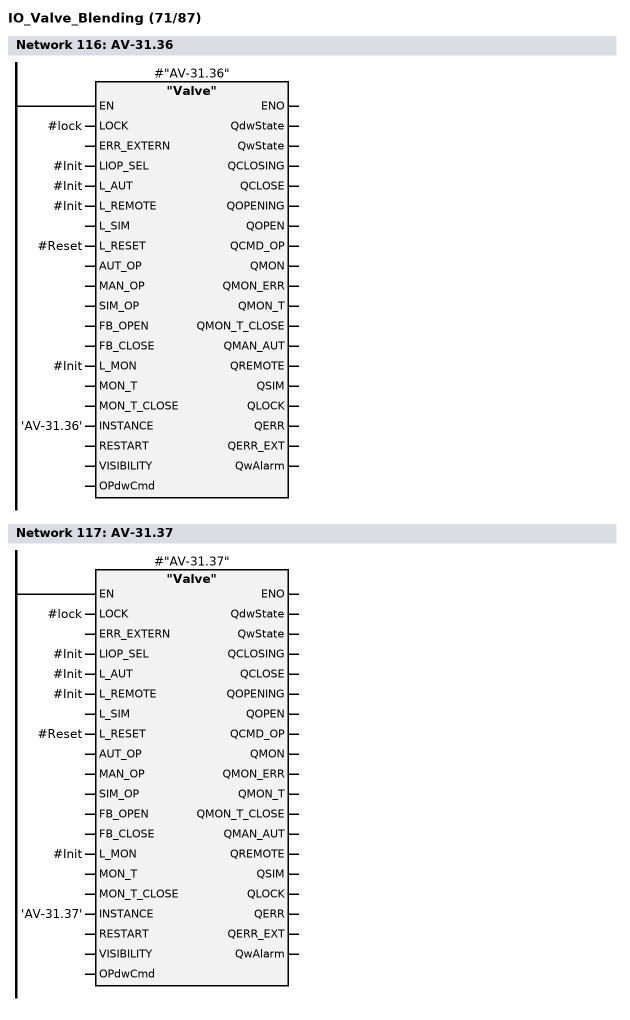
   RUNG wire#powerrail
      #"AV-31.36"(LOCK := #lock, ERR_EXTERN :=, LIOP_SEL := #Init, L_AUT := #Init, L_REMOTE := #Init, L_SIM :=, L_RESET := #Reset, AUT_OP :=, MAN_OP :=, SIM_OP :=, FB_OPEN :=, FB_CLOSE :=, L_MON := #Init, MON_T :=, MON_T_CLOSE :=, INSTANCE := 'AV-31.36', RESTART :=, VISIBILITY :=, OPdwCmd :=, QdwState =>, QwState =>, QCLOSING =>, QCLOSE =>, QOPENING =>, QOPEN =>, QCMD_OP =>, QMON =>, QMON_ERR =>, QMON_T =>, QMON_T_CLOSE =>, QMAN_AUT =>, QREMOTE =>, QSIM =>, QLOCK =>, QERR =>, QERR_EXT =>, QwAlarm =>)
   END_RUNG
   // the same network as SCL:
   #"AV-31.36"(LOCK := #lock,   // "Valve"
               LIOP_SEL := #Init,
               L_AUT := #Init,
               L_REMOTE := #Init,
               L_RESET := #Reset,
               L_MON := #Init,
               INSTANCE := 'AV-31.36');
END_REGION

REGION Network 117: AV-31.37
   RUNG wire#powerrail
      #"AV-31.37"(LOCK := #lock, ERR_EXTERN :=, LIOP_SEL := #Init, L_AUT := #Init, L_REMOTE := #Init, L_SIM :=, L_RESET := #Reset, AUT_OP :=, MAN_OP :=, SIM_OP :=, FB_OPEN :=, FB_CLOSE :=, L_MON := #Init, MON_T :=, MON_T_CLOSE :=, INSTANCE := 'AV-31.37', RESTART :=, VISIBILITY :=, OPdwCmd :=, QdwState =>, QwState =>, QCLOSING =>, QCLOSE =>, QOPENING =>, QOPEN =>, QCMD_OP =>, QMON =>, QMON_ERR =>, QMON_T =>, QMON_T_CLOSE =>, QMAN_AUT =>, QREMOTE =>, QSIM =>, QLOCK =>, QERR =>, QERR_EXT =>, QwAlarm =>)
   END_RUNG
   // the same network as SCL:
   #"AV-31.37"(LOCK := #lock,   // "Valve"
               LIOP_SEL := #Init,
               L_AUT := #Init,
               L_REMOTE := #Init,
               L_RESET := #Reset,
               L_MON := #Init,
               INSTANCE := 'AV-31.37');
END_REGION

REGION Network 118: AV-31.38
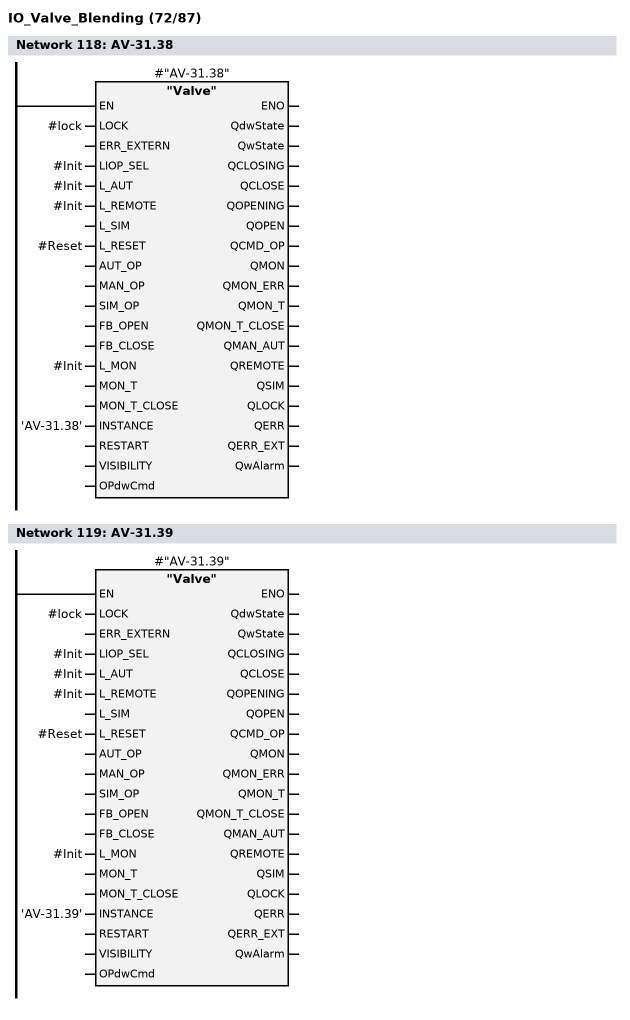
   RUNG wire#powerrail
      #"AV-31.38"(LOCK := #lock, ERR_EXTERN :=, LIOP_SEL := #Init, L_AUT := #Init, L_REMOTE := #Init, L_SIM :=, L_RESET := #Reset, AUT_OP :=, MAN_OP :=, SIM_OP :=, FB_OPEN :=, FB_CLOSE :=, L_MON := #Init, MON_T :=, MON_T_CLOSE :=, INSTANCE := 'AV-31.38', RESTART :=, VISIBILITY :=, OPdwCmd :=, QdwState =>, QwState =>, QCLOSING =>, QCLOSE =>, QOPENING =>, QOPEN =>, QCMD_OP =>, QMON =>, QMON_ERR =>, QMON_T =>, QMON_T_CLOSE =>, QMAN_AUT =>, QREMOTE =>, QSIM =>, QLOCK =>, QERR =>, QERR_EXT =>, QwAlarm =>)
   END_RUNG
   // the same network as SCL:
   #"AV-31.38"(LOCK := #lock,   // "Valve"
               LIOP_SEL := #Init,
               L_AUT := #Init,
               L_REMOTE := #Init,
               L_RESET := #Reset,
               L_MON := #Init,
               INSTANCE := 'AV-31.38');
END_REGION

REGION Network 119: AV-31.39
   RUNG wire#powerrail
      #"AV-31.39"(LOCK := #lock, ERR_EXTERN :=, LIOP_SEL := #Init, L_AUT := #Init, L_REMOTE := #Init, L_SIM :=, L_RESET := #Reset, AUT_OP :=, MAN_OP :=, SIM_OP :=, FB_OPEN :=, FB_CLOSE :=, L_MON := #Init, MON_T :=, MON_T_CLOSE :=, INSTANCE := 'AV-31.39', RESTART :=, VISIBILITY :=, OPdwCmd :=, QdwState =>, QwState =>, QCLOSING =>, QCLOSE =>, QOPENING =>, QOPEN =>, QCMD_OP =>, QMON =>, QMON_ERR =>, QMON_T =>, QMON_T_CLOSE =>, QMAN_AUT =>, QREMOTE =>, QSIM =>, QLOCK =>, QERR =>, QERR_EXT =>, QwAlarm =>)
   END_RUNG
   // the same network as SCL:
   #"AV-31.39"(LOCK := #lock,   // "Valve"
               LIOP_SEL := #Init,
               L_AUT := #Init,
               L_REMOTE := #Init,
               L_RESET := #Reset,
               L_MON := #Init,
               INSTANCE := 'AV-31.39');
END_REGION

REGION Network 120: AV-31.40
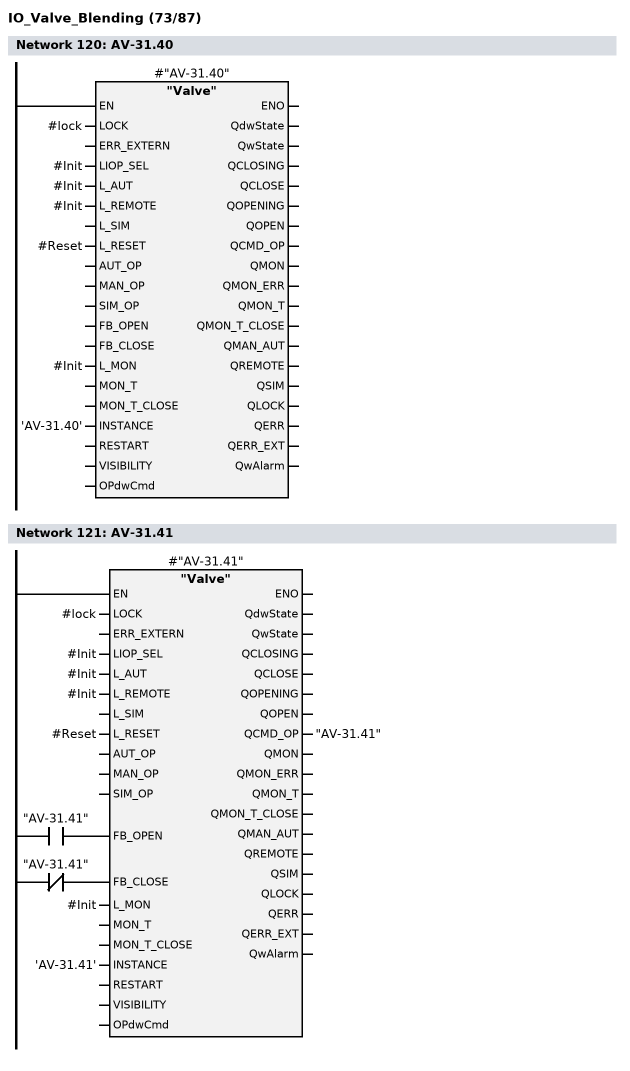
   RUNG wire#powerrail
      #"AV-31.40"(LOCK := #lock, ERR_EXTERN :=, LIOP_SEL := #Init, L_AUT := #Init, L_REMOTE := #Init, L_SIM :=, L_RESET := #Reset, AUT_OP :=, MAN_OP :=, SIM_OP :=, FB_OPEN :=, FB_CLOSE :=, L_MON := #Init, MON_T :=, MON_T_CLOSE :=, INSTANCE := 'AV-31.40', RESTART :=, VISIBILITY :=, OPdwCmd :=, QdwState =>, QwState =>, QCLOSING =>, QCLOSE =>, QOPENING =>, QOPEN =>, QCMD_OP =>, QMON =>, QMON_ERR =>, QMON_T =>, QMON_T_CLOSE =>, QMAN_AUT =>, QREMOTE =>, QSIM =>, QLOCK =>, QERR =>, QERR_EXT =>, QwAlarm =>)
   END_RUNG
   // the same network as SCL:
   #"AV-31.40"(LOCK := #lock,   // "Valve"
               LIOP_SEL := #Init,
               L_AUT := #Init,
               L_REMOTE := #Init,
               L_RESET := #Reset,
               L_MON := #Init,
               INSTANCE := 'AV-31.40');
END_REGION

REGION Network 121: AV-31.41
   RUNG wire#powerrail
      #"AV-31.41"(FB_OPEN := wire#w1, FB_CLOSE := wire#w2, LOCK := #lock, ERR_EXTERN :=, LIOP_SEL := #Init, L_AUT := #Init, L_REMOTE := #Init, L_SIM :=, L_RESET := #Reset, AUT_OP :=, MAN_OP :=, SIM_OP :=, L_MON := #Init, MON_T :=, MON_T_CLOSE :=, INSTANCE := 'AV-31.41', RESTART :=, VISIBILITY :=, OPdwCmd :=, QdwState =>, QwState =>, QCLOSING =>, QCLOSE =>, QOPENING =>, QOPEN =>, QCMD_OP => "AV-31.41", QMON =>, QMON_ERR =>, QMON_T =>, QMON_T_CLOSE =>, QMAN_AUT =>, QREMOTE =>, QSIM =>, QLOCK =>, QERR =>, QERR_EXT =>, QwAlarm =>)
   END_RUNG
   RUNG wire#powerrail
      Contact( "AV-31.41" )
   END_RUNG wire#w1
   RUNG wire#powerrail
      I_Contact( "AV-31.41" )
   END_RUNG wire#w2
   // the same network as SCL:
   #"AV-31.41"(LOCK := #lock,   // "Valve"
               LIOP_SEL := #Init,
               L_AUT := #Init,
               L_REMOTE := #Init,
               L_RESET := #Reset,
               FB_OPEN := "AV-31.41",
               FB_CLOSE := NOT "AV-31.41",
               L_MON := #Init,
               INSTANCE := 'AV-31.41',
               QCMD_OP => "AV-31.41");
END_REGION

REGION Network 122: AV-31.51
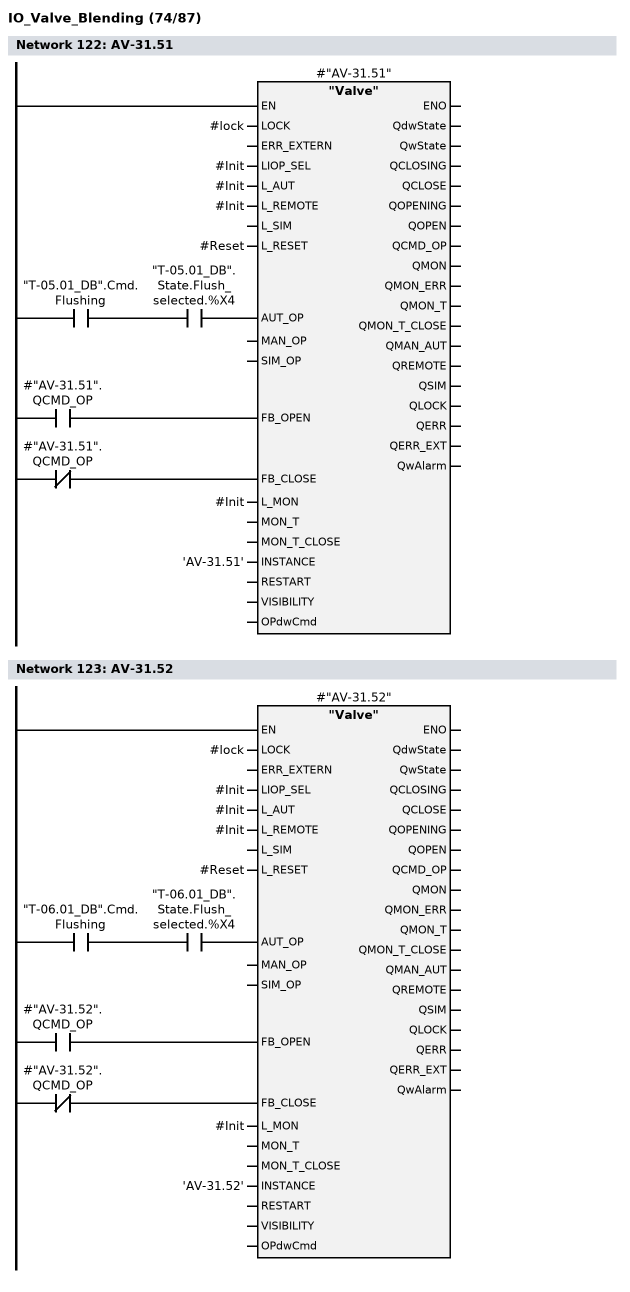
   RUNG wire#powerrail
      #"AV-31.51"(AUT_OP := wire#w1, FB_OPEN := wire#w2, FB_CLOSE := wire#w3, LOCK := #lock, ERR_EXTERN :=, LIOP_SEL := #Init, L_AUT := #Init, L_REMOTE := #Init, L_SIM :=, L_RESET := #Reset, MAN_OP :=, SIM_OP :=, L_MON := #Init, MON_T :=, MON_T_CLOSE :=, INSTANCE := 'AV-31.51', RESTART :=, VISIBILITY :=, OPdwCmd :=, QdwState =>, QwState =>, QCLOSING =>, QCLOSE =>, QOPENING =>, QOPEN =>, QCMD_OP =>, QMON =>, QMON_ERR =>, QMON_T =>, QMON_T_CLOSE =>, QMAN_AUT =>, QREMOTE =>, QSIM =>, QLOCK =>, QERR =>, QERR_EXT =>, QwAlarm =>)
   END_RUNG
   RUNG wire#powerrail
      Contact( "T-05.01_DB".Cmd.Flushing )
      Contact( "T-05.01_DB".State.Flush_selected.%X4 )
   END_RUNG wire#w1
   RUNG wire#powerrail
      Contact( #"AV-31.51".QCMD_OP )
   END_RUNG wire#w2
   RUNG wire#powerrail
      I_Contact( #"AV-31.51".QCMD_OP )
   END_RUNG wire#w3
   // the same network as SCL:
   #"AV-31.51"(LOCK := #lock,   // "Valve"
               LIOP_SEL := #Init,
               L_AUT := #Init,
               L_REMOTE := #Init,
               L_RESET := #Reset,
               AUT_OP := "T-05.01_DB".Cmd.Flushing AND "T-05.01_DB".State.Flush_selected.%X4,
               FB_OPEN := #"AV-31.51".QCMD_OP,
               FB_CLOSE := NOT #"AV-31.51".QCMD_OP,
               L_MON := #Init,
               INSTANCE := 'AV-31.51');
END_REGION

REGION Network 123: AV-31.52
   RUNG wire#powerrail
      #"AV-31.52"(AUT_OP := wire#w1, FB_OPEN := wire#w2, FB_CLOSE := wire#w3, LOCK := #lock, ERR_EXTERN :=, LIOP_SEL := #Init, L_AUT := #Init, L_REMOTE := #Init, L_SIM :=, L_RESET := #Reset, MAN_OP :=, SIM_OP :=, L_MON := #Init, MON_T :=, MON_T_CLOSE :=, INSTANCE := 'AV-31.52', RESTART :=, VISIBILITY :=, OPdwCmd :=, QdwState =>, QwState =>, QCLOSING =>, QCLOSE =>, QOPENING =>, QOPEN =>, QCMD_OP =>, QMON =>, QMON_ERR =>, QMON_T =>, QMON_T_CLOSE =>, QMAN_AUT =>, QREMOTE =>, QSIM =>, QLOCK =>, QERR =>, QERR_EXT =>, QwAlarm =>)
   END_RUNG
   RUNG wire#powerrail
      Contact( "T-06.01_DB".Cmd.Flushing )
      Contact( "T-06.01_DB".State.Flush_selected.%X4 )
   END_RUNG wire#w1
   RUNG wire#powerrail
      Contact( #"AV-31.52".QCMD_OP )
   END_RUNG wire#w2
   RUNG wire#powerrail
      I_Contact( #"AV-31.52".QCMD_OP )
   END_RUNG wire#w3
   // the same network as SCL:
   #"AV-31.52"(LOCK := #lock,   // "Valve"
               LIOP_SEL := #Init,
               L_AUT := #Init,
               L_REMOTE := #Init,
               L_RESET := #Reset,
               AUT_OP := "T-06.01_DB".Cmd.Flushing AND "T-06.01_DB".State.Flush_selected.%X4,
               FB_OPEN := #"AV-31.52".QCMD_OP,
               FB_CLOSE := NOT #"AV-31.52".QCMD_OP,
               L_MON := #Init,
               INSTANCE := 'AV-31.52');
END_REGION

REGION Network 124: AV-31.53
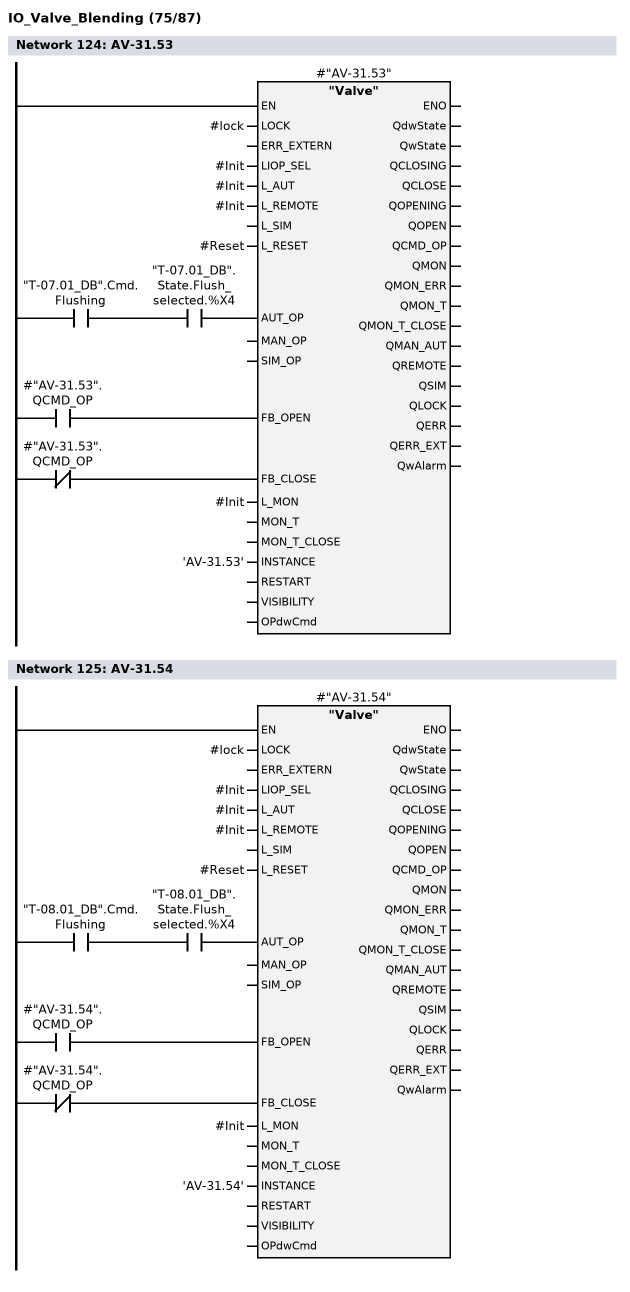
   RUNG wire#powerrail
      #"AV-31.53"(AUT_OP := wire#w1, FB_OPEN := wire#w2, FB_CLOSE := wire#w3, LOCK := #lock, ERR_EXTERN :=, LIOP_SEL := #Init, L_AUT := #Init, L_REMOTE := #Init, L_SIM :=, L_RESET := #Reset, MAN_OP :=, SIM_OP :=, L_MON := #Init, MON_T :=, MON_T_CLOSE :=, INSTANCE := 'AV-31.53', RESTART :=, VISIBILITY :=, OPdwCmd :=, QdwState =>, QwState =>, QCLOSING =>, QCLOSE =>, QOPENING =>, QOPEN =>, QCMD_OP =>, QMON =>, QMON_ERR =>, QMON_T =>, QMON_T_CLOSE =>, QMAN_AUT =>, QREMOTE =>, QSIM =>, QLOCK =>, QERR =>, QERR_EXT =>, QwAlarm =>)
   END_RUNG
   RUNG wire#powerrail
      Contact( "T-07.01_DB".Cmd.Flushing )
      Contact( "T-07.01_DB".State.Flush_selected.%X4 )
   END_RUNG wire#w1
   RUNG wire#powerrail
      Contact( #"AV-31.53".QCMD_OP )
   END_RUNG wire#w2
   RUNG wire#powerrail
      I_Contact( #"AV-31.53".QCMD_OP )
   END_RUNG wire#w3
   // the same network as SCL:
   #"AV-31.53"(LOCK := #lock,   // "Valve"
               LIOP_SEL := #Init,
               L_AUT := #Init,
               L_REMOTE := #Init,
               L_RESET := #Reset,
               AUT_OP := "T-07.01_DB".Cmd.Flushing AND "T-07.01_DB".State.Flush_selected.%X4,
               FB_OPEN := #"AV-31.53".QCMD_OP,
               FB_CLOSE := NOT #"AV-31.53".QCMD_OP,
               L_MON := #Init,
               INSTANCE := 'AV-31.53');
END_REGION

REGION Network 125: AV-31.54
   RUNG wire#powerrail
      #"AV-31.54"(AUT_OP := wire#w1, FB_OPEN := wire#w2, FB_CLOSE := wire#w3, LOCK := #lock, ERR_EXTERN :=, LIOP_SEL := #Init, L_AUT := #Init, L_REMOTE := #Init, L_SIM :=, L_RESET := #Reset, MAN_OP :=, SIM_OP :=, L_MON := #Init, MON_T :=, MON_T_CLOSE :=, INSTANCE := 'AV-31.54', RESTART :=, VISIBILITY :=, OPdwCmd :=, QdwState =>, QwState =>, QCLOSING =>, QCLOSE =>, QOPENING =>, QOPEN =>, QCMD_OP =>, QMON =>, QMON_ERR =>, QMON_T =>, QMON_T_CLOSE =>, QMAN_AUT =>, QREMOTE =>, QSIM =>, QLOCK =>, QERR =>, QERR_EXT =>, QwAlarm =>)
   END_RUNG
   RUNG wire#powerrail
      Contact( "T-08.01_DB".Cmd.Flushing )
      Contact( "T-08.01_DB".State.Flush_selected.%X4 )
   END_RUNG wire#w1
   RUNG wire#powerrail
      Contact( #"AV-31.54".QCMD_OP )
   END_RUNG wire#w2
   RUNG wire#powerrail
      I_Contact( #"AV-31.54".QCMD_OP )
   END_RUNG wire#w3
   // the same network as SCL:
   #"AV-31.54"(LOCK := #lock,   // "Valve"
               LIOP_SEL := #Init,
               L_AUT := #Init,
               L_REMOTE := #Init,
               L_RESET := #Reset,
               AUT_OP := "T-08.01_DB".Cmd.Flushing AND "T-08.01_DB".State.Flush_selected.%X4,
               FB_OPEN := #"AV-31.54".QCMD_OP,
               FB_CLOSE := NOT #"AV-31.54".QCMD_OP,
               L_MON := #Init,
               INSTANCE := 'AV-31.54');
END_REGION

REGION Network 126: AV-31.55
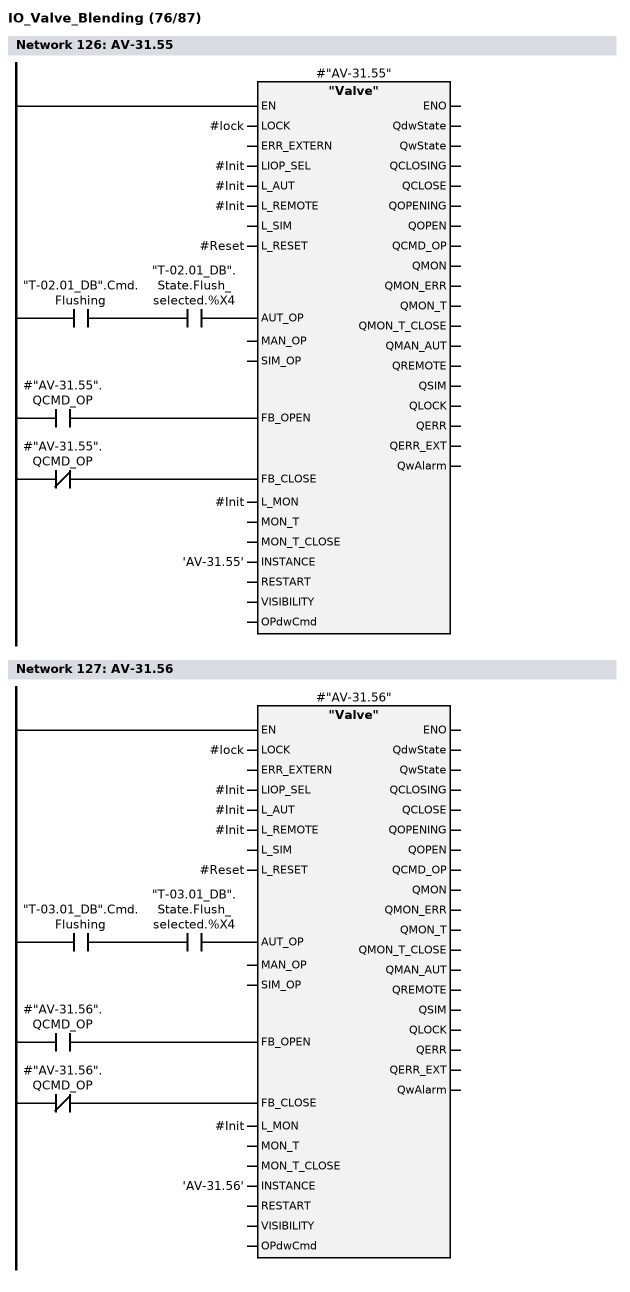
   RUNG wire#powerrail
      #"AV-31.55"(AUT_OP := wire#w1, FB_OPEN := wire#w2, FB_CLOSE := wire#w3, LOCK := #lock, ERR_EXTERN :=, LIOP_SEL := #Init, L_AUT := #Init, L_REMOTE := #Init, L_SIM :=, L_RESET := #Reset, MAN_OP :=, SIM_OP :=, L_MON := #Init, MON_T :=, MON_T_CLOSE :=, INSTANCE := 'AV-31.55', RESTART :=, VISIBILITY :=, OPdwCmd :=, QdwState =>, QwState =>, QCLOSING =>, QCLOSE =>, QOPENING =>, QOPEN =>, QCMD_OP =>, QMON =>, QMON_ERR =>, QMON_T =>, QMON_T_CLOSE =>, QMAN_AUT =>, QREMOTE =>, QSIM =>, QLOCK =>, QERR =>, QERR_EXT =>, QwAlarm =>)
   END_RUNG
   RUNG wire#powerrail
      Contact( "T-02.01_DB".Cmd.Flushing )
      Contact( "T-02.01_DB".State.Flush_selected.%X4 )
   END_RUNG wire#w1
   RUNG wire#powerrail
      Contact( #"AV-31.55".QCMD_OP )
   END_RUNG wire#w2
   RUNG wire#powerrail
      I_Contact( #"AV-31.55".QCMD_OP )
   END_RUNG wire#w3
   // the same network as SCL:
   #"AV-31.55"(LOCK := #lock,   // "Valve"
               LIOP_SEL := #Init,
               L_AUT := #Init,
               L_REMOTE := #Init,
               L_RESET := #Reset,
               AUT_OP := "T-02.01_DB".Cmd.Flushing AND "T-02.01_DB".State.Flush_selected.%X4,
               FB_OPEN := #"AV-31.55".QCMD_OP,
               FB_CLOSE := NOT #"AV-31.55".QCMD_OP,
               L_MON := #Init,
               INSTANCE := 'AV-31.55');
END_REGION

REGION Network 127: AV-31.56
   RUNG wire#powerrail
      #"AV-31.56"(AUT_OP := wire#w1, FB_OPEN := wire#w2, FB_CLOSE := wire#w3, LOCK := #lock, ERR_EXTERN :=, LIOP_SEL := #Init, L_AUT := #Init, L_REMOTE := #Init, L_SIM :=, L_RESET := #Reset, MAN_OP :=, SIM_OP :=, L_MON := #Init, MON_T :=, MON_T_CLOSE :=, INSTANCE := 'AV-31.56', RESTART :=, VISIBILITY :=, OPdwCmd :=, QdwState =>, QwState =>, QCLOSING =>, QCLOSE =>, QOPENING =>, QOPEN =>, QCMD_OP =>, QMON =>, QMON_ERR =>, QMON_T =>, QMON_T_CLOSE =>, QMAN_AUT =>, QREMOTE =>, QSIM =>, QLOCK =>, QERR =>, QERR_EXT =>, QwAlarm =>)
   END_RUNG
   RUNG wire#powerrail
      Contact( "T-03.01_DB".Cmd.Flushing )
      Contact( "T-03.01_DB".State.Flush_selected.%X4 )
   END_RUNG wire#w1
   RUNG wire#powerrail
      Contact( #"AV-31.56".QCMD_OP )
   END_RUNG wire#w2
   RUNG wire#powerrail
      I_Contact( #"AV-31.56".QCMD_OP )
   END_RUNG wire#w3
   // the same network as SCL:
   #"AV-31.56"(LOCK := #lock,   // "Valve"
               LIOP_SEL := #Init,
               L_AUT := #Init,
               L_REMOTE := #Init,
               L_RESET := #Reset,
               AUT_OP := "T-03.01_DB".Cmd.Flushing AND "T-03.01_DB".State.Flush_selected.%X4,
               FB_OPEN := #"AV-31.56".QCMD_OP,
               FB_CLOSE := NOT #"AV-31.56".QCMD_OP,
               L_MON := #Init,
               INSTANCE := 'AV-31.56');
END_REGION

REGION Network 128: AV-31.57
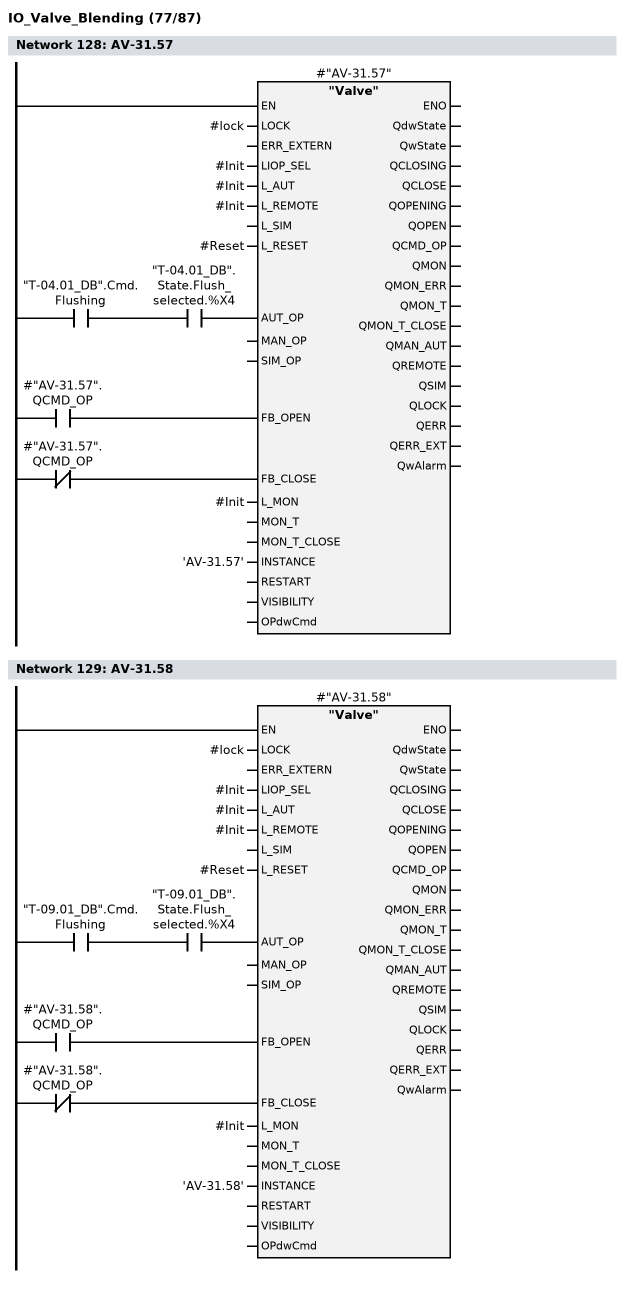
   RUNG wire#powerrail
      #"AV-31.57"(AUT_OP := wire#w1, FB_OPEN := wire#w2, FB_CLOSE := wire#w3, LOCK := #lock, ERR_EXTERN :=, LIOP_SEL := #Init, L_AUT := #Init, L_REMOTE := #Init, L_SIM :=, L_RESET := #Reset, MAN_OP :=, SIM_OP :=, L_MON := #Init, MON_T :=, MON_T_CLOSE :=, INSTANCE := 'AV-31.57', RESTART :=, VISIBILITY :=, OPdwCmd :=, QdwState =>, QwState =>, QCLOSING =>, QCLOSE =>, QOPENING =>, QOPEN =>, QCMD_OP =>, QMON =>, QMON_ERR =>, QMON_T =>, QMON_T_CLOSE =>, QMAN_AUT =>, QREMOTE =>, QSIM =>, QLOCK =>, QERR =>, QERR_EXT =>, QwAlarm =>)
   END_RUNG
   RUNG wire#powerrail
      Contact( "T-04.01_DB".Cmd.Flushing )
      Contact( "T-04.01_DB".State.Flush_selected.%X4 )
   END_RUNG wire#w1
   RUNG wire#powerrail
      Contact( #"AV-31.57".QCMD_OP )
   END_RUNG wire#w2
   RUNG wire#powerrail
      I_Contact( #"AV-31.57".QCMD_OP )
   END_RUNG wire#w3
   // the same network as SCL:
   #"AV-31.57"(LOCK := #lock,   // "Valve"
               LIOP_SEL := #Init,
               L_AUT := #Init,
               L_REMOTE := #Init,
               L_RESET := #Reset,
               AUT_OP := "T-04.01_DB".Cmd.Flushing AND "T-04.01_DB".State.Flush_selected.%X4,
               FB_OPEN := #"AV-31.57".QCMD_OP,
               FB_CLOSE := NOT #"AV-31.57".QCMD_OP,
               L_MON := #Init,
               INSTANCE := 'AV-31.57');
END_REGION

REGION Network 129: AV-31.58
   RUNG wire#powerrail
      #"AV-31.58"(AUT_OP := wire#w1, FB_OPEN := wire#w2, FB_CLOSE := wire#w3, LOCK := #lock, ERR_EXTERN :=, LIOP_SEL := #Init, L_AUT := #Init, L_REMOTE := #Init, L_SIM :=, L_RESET := #Reset, MAN_OP :=, SIM_OP :=, L_MON := #Init, MON_T :=, MON_T_CLOSE :=, INSTANCE := 'AV-31.58', RESTART :=, VISIBILITY :=, OPdwCmd :=, QdwState =>, QwState =>, QCLOSING =>, QCLOSE =>, QOPENING =>, QOPEN =>, QCMD_OP =>, QMON =>, QMON_ERR =>, QMON_T =>, QMON_T_CLOSE =>, QMAN_AUT =>, QREMOTE =>, QSIM =>, QLOCK =>, QERR =>, QERR_EXT =>, QwAlarm =>)
   END_RUNG
   RUNG wire#powerrail
      Contact( "T-09.01_DB".Cmd.Flushing )
      Contact( "T-09.01_DB".State.Flush_selected.%X4 )
   END_RUNG wire#w1
   RUNG wire#powerrail
      Contact( #"AV-31.58".QCMD_OP )
   END_RUNG wire#w2
   RUNG wire#powerrail
      I_Contact( #"AV-31.58".QCMD_OP )
   END_RUNG wire#w3
   // the same network as SCL:
   #"AV-31.58"(LOCK := #lock,   // "Valve"
               LIOP_SEL := #Init,
               L_AUT := #Init,
               L_REMOTE := #Init,
               L_RESET := #Reset,
               AUT_OP := "T-09.01_DB".Cmd.Flushing AND "T-09.01_DB".State.Flush_selected.%X4,
               FB_OPEN := #"AV-31.58".QCMD_OP,
               FB_CLOSE := NOT #"AV-31.58".QCMD_OP,
               L_MON := #Init,
               INSTANCE := 'AV-31.58');
END_REGION

REGION Network 130: AV-31.59
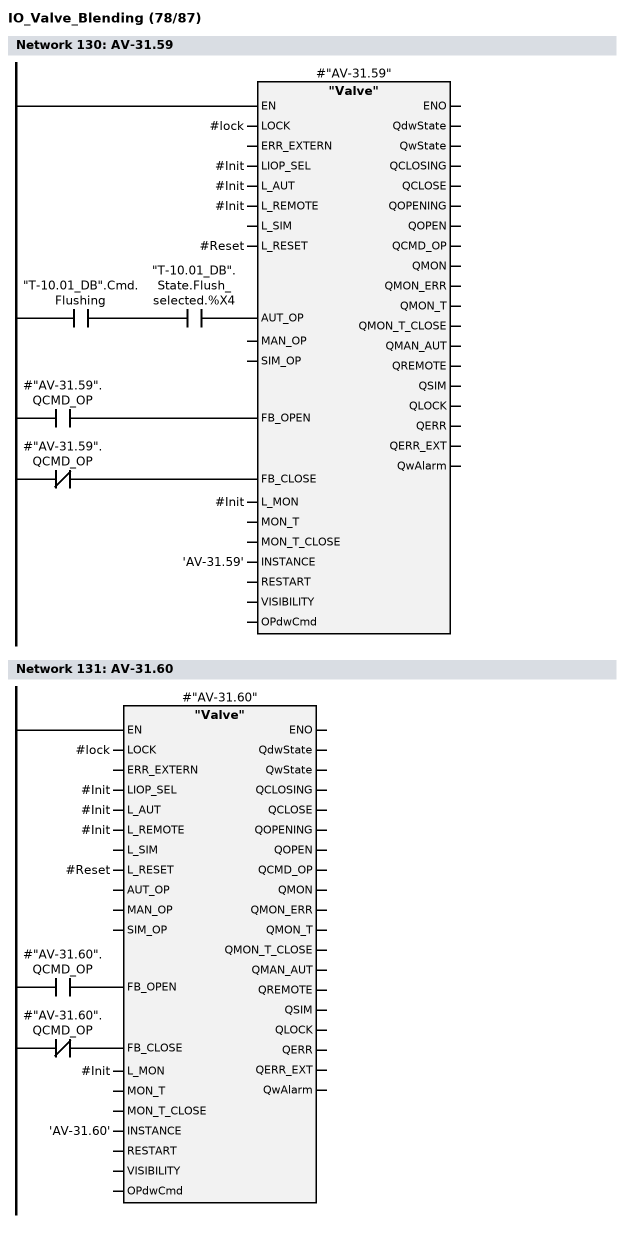
   RUNG wire#powerrail
      #"AV-31.59"(AUT_OP := wire#w1, FB_OPEN := wire#w2, FB_CLOSE := wire#w3, LOCK := #lock, ERR_EXTERN :=, LIOP_SEL := #Init, L_AUT := #Init, L_REMOTE := #Init, L_SIM :=, L_RESET := #Reset, MAN_OP :=, SIM_OP :=, L_MON := #Init, MON_T :=, MON_T_CLOSE :=, INSTANCE := 'AV-31.59', RESTART :=, VISIBILITY :=, OPdwCmd :=, QdwState =>, QwState =>, QCLOSING =>, QCLOSE =>, QOPENING =>, QOPEN =>, QCMD_OP =>, QMON =>, QMON_ERR =>, QMON_T =>, QMON_T_CLOSE =>, QMAN_AUT =>, QREMOTE =>, QSIM =>, QLOCK =>, QERR =>, QERR_EXT =>, QwAlarm =>)
   END_RUNG
   RUNG wire#powerrail
      Contact( "T-10.01_DB".Cmd.Flushing )
      Contact( "T-10.01_DB".State.Flush_selected.%X4 )
   END_RUNG wire#w1
   RUNG wire#powerrail
      Contact( #"AV-31.59".QCMD_OP )
   END_RUNG wire#w2
   RUNG wire#powerrail
      I_Contact( #"AV-31.59".QCMD_OP )
   END_RUNG wire#w3
   // the same network as SCL:
   #"AV-31.59"(LOCK := #lock,   // "Valve"
               LIOP_SEL := #Init,
               L_AUT := #Init,
               L_REMOTE := #Init,
               L_RESET := #Reset,
               AUT_OP := "T-10.01_DB".Cmd.Flushing AND "T-10.01_DB".State.Flush_selected.%X4,
               FB_OPEN := #"AV-31.59".QCMD_OP,
               FB_CLOSE := NOT #"AV-31.59".QCMD_OP,
               L_MON := #Init,
               INSTANCE := 'AV-31.59');
END_REGION

REGION Network 131: AV-31.60
   RUNG wire#powerrail
      #"AV-31.60"(FB_OPEN := wire#w1, FB_CLOSE := wire#w2, LOCK := #lock, ERR_EXTERN :=, LIOP_SEL := #Init, L_AUT := #Init, L_REMOTE := #Init, L_SIM :=, L_RESET := #Reset, AUT_OP :=, MAN_OP :=, SIM_OP :=, L_MON := #Init, MON_T :=, MON_T_CLOSE :=, INSTANCE := 'AV-31.60', RESTART :=, VISIBILITY :=, OPdwCmd :=, QdwState =>, QwState =>, QCLOSING =>, QCLOSE =>, QOPENING =>, QOPEN =>, QCMD_OP =>, QMON =>, QMON_ERR =>, QMON_T =>, QMON_T_CLOSE =>, QMAN_AUT =>, QREMOTE =>, QSIM =>, QLOCK =>, QERR =>, QERR_EXT =>, QwAlarm =>)
   END_RUNG
   RUNG wire#powerrail
      Contact( #"AV-31.60".QCMD_OP )
   END_RUNG wire#w1
   RUNG wire#powerrail
      I_Contact( #"AV-31.60".QCMD_OP )
   END_RUNG wire#w2
   // the same network as SCL:
   #"AV-31.60"(LOCK := #lock,   // "Valve"
               LIOP_SEL := #Init,
               L_AUT := #Init,
               L_REMOTE := #Init,
               L_RESET := #Reset,
               FB_OPEN := #"AV-31.60".QCMD_OP,
               FB_CLOSE := NOT #"AV-31.60".QCMD_OP,
               L_MON := #Init,
               INSTANCE := 'AV-31.60');
END_REGION

REGION Network 132: AV-31.61
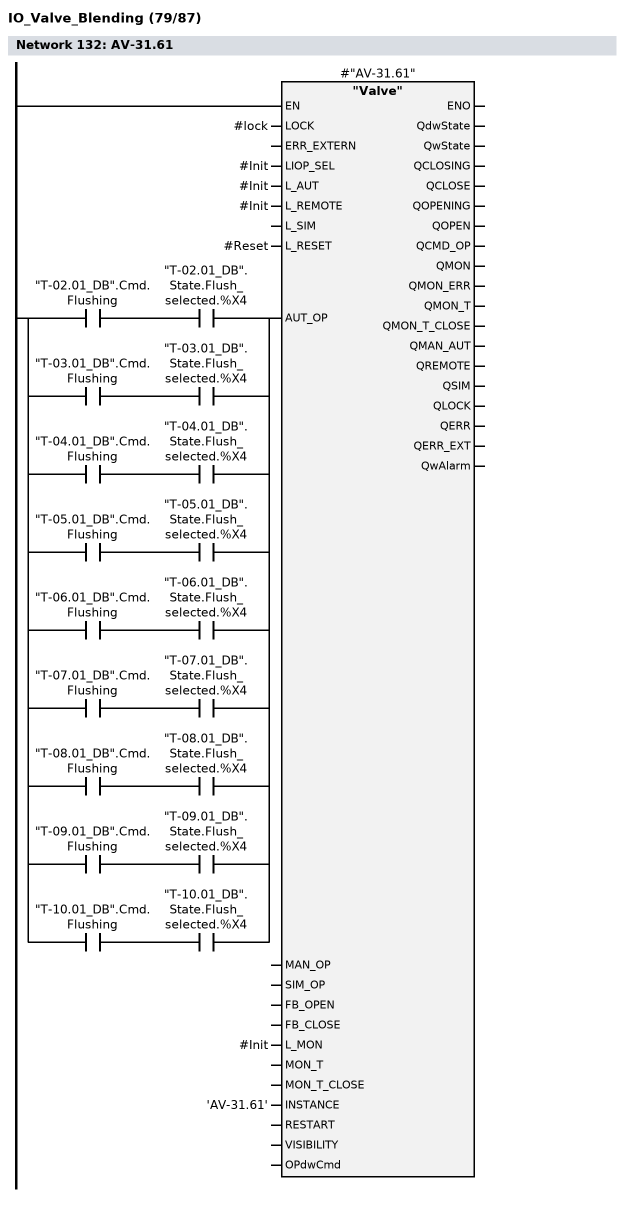
   RUNG wire#powerrail
      #"AV-31.61"(AUT_OP := wire#w1, LOCK := #lock, ERR_EXTERN :=, LIOP_SEL := #Init, L_AUT := #Init, L_REMOTE := #Init, L_SIM :=, L_RESET := #Reset, MAN_OP :=, SIM_OP :=, FB_OPEN :=, FB_CLOSE :=, L_MON := #Init, MON_T :=, MON_T_CLOSE :=, INSTANCE := 'AV-31.61', RESTART :=, VISIBILITY :=, OPdwCmd :=, QdwState =>, QwState =>, QCLOSING =>, QCLOSE =>, QOPENING =>, QOPEN =>, QCMD_OP =>, QMON =>, QMON_ERR =>, QMON_T =>, QMON_T_CLOSE =>, QMAN_AUT =>, QREMOTE =>, QSIM =>, QLOCK =>, QERR =>, QERR_EXT =>, QwAlarm =>)
   END_RUNG
   RUNG wire#powerrail
      Contact( "T-02.01_DB".Cmd.Flushing )
      Contact( "T-02.01_DB".State.Flush_selected.%X4 )
   END_RUNG wire#w1
   RUNG wire#powerrail
      Contact( "T-03.01_DB".Cmd.Flushing )
      Contact( "T-03.01_DB".State.Flush_selected.%X4 )
   END_RUNG wire#w1
   RUNG wire#powerrail
      Contact( "T-04.01_DB".Cmd.Flushing )
      Contact( "T-04.01_DB".State.Flush_selected.%X4 )
   END_RUNG wire#w1
   RUNG wire#powerrail
      Contact( "T-05.01_DB".Cmd.Flushing )
      Contact( "T-05.01_DB".State.Flush_selected.%X4 )
   END_RUNG wire#w1
   RUNG wire#powerrail
      Contact( "T-06.01_DB".Cmd.Flushing )
      Contact( "T-06.01_DB".State.Flush_selected.%X4 )
   END_RUNG wire#w1
   RUNG wire#powerrail
      Contact( "T-07.01_DB".Cmd.Flushing )
      Contact( "T-07.01_DB".State.Flush_selected.%X4 )
   END_RUNG wire#w1
   RUNG wire#powerrail
      Contact( "T-08.01_DB".Cmd.Flushing )
      Contact( "T-08.01_DB".State.Flush_selected.%X4 )
   END_RUNG wire#w1
   RUNG wire#powerrail
      Contact( "T-09.01_DB".Cmd.Flushing )
      Contact( "T-09.01_DB".State.Flush_selected.%X4 )
   END_RUNG wire#w1
   RUNG wire#powerrail
      Contact( "T-10.01_DB".Cmd.Flushing )
      Contact( "T-10.01_DB".State.Flush_selected.%X4 )
   END_RUNG wire#w1
   // the same network as SCL:
   #"AV-31.61"(LOCK := #lock,   // "Valve"
               LIOP_SEL := #Init,
               L_AUT := #Init,
               L_REMOTE := #Init,
               L_RESET := #Reset,
               AUT_OP := ("T-02.01_DB".Cmd.Flushing AND "T-02.01_DB".State.Flush_selected.%X4) OR ("T-03.01_DB".Cmd.Flushing AND "T-03.01_DB".State.Flush_selected.%X4) OR ("T-04.01_DB".Cmd.Flushing AND "T-04.01_DB".State.Flush_selected.%X4) OR ("T-05.01_DB".Cmd.Flushing AND "T-05.01_DB".State.Flush_selected.%X4) OR ("T-06.01_DB".Cmd.Flushing AND "T-06.01_DB".State.Flush_selected.%X4) OR ("T-07.01_DB".Cmd.Flushing AND "T-07.01_DB".State.Flush_selected.%X4) OR ("T-08.01_DB".Cmd.Flushing AND "T-08.01_DB".State.Flush_selected.%X4) OR ("T-09.01_DB".Cmd.Flushing AND "T-09.01_DB".State.Flush_selected.%X4) OR ("T-10.01_DB".Cmd.Flushing AND "T-10.01_DB".State.Flush_selected.%X4),
               L_MON := #Init,
               INSTANCE := 'AV-31.61');
END_REGION

REGION Network 133: AV-31.62
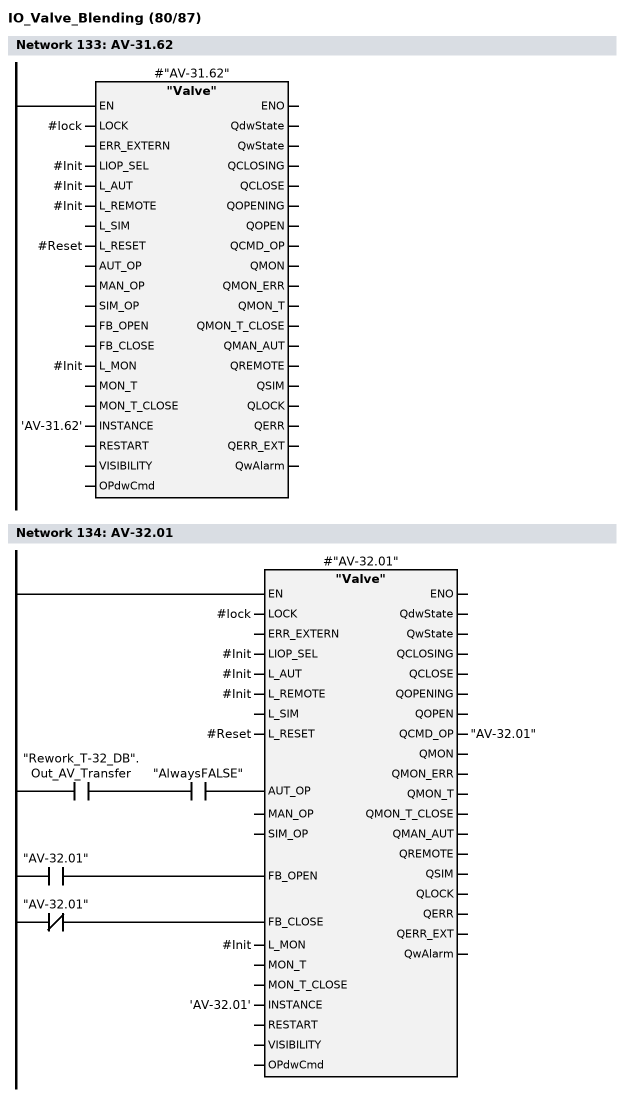
   RUNG wire#powerrail
      #"AV-31.62"(LOCK := #lock, ERR_EXTERN :=, LIOP_SEL := #Init, L_AUT := #Init, L_REMOTE := #Init, L_SIM :=, L_RESET := #Reset, AUT_OP :=, MAN_OP :=, SIM_OP :=, FB_OPEN :=, FB_CLOSE :=, L_MON := #Init, MON_T :=, MON_T_CLOSE :=, INSTANCE := 'AV-31.62', RESTART :=, VISIBILITY :=, OPdwCmd :=, QdwState =>, QwState =>, QCLOSING =>, QCLOSE =>, QOPENING =>, QOPEN =>, QCMD_OP =>, QMON =>, QMON_ERR =>, QMON_T =>, QMON_T_CLOSE =>, QMAN_AUT =>, QREMOTE =>, QSIM =>, QLOCK =>, QERR =>, QERR_EXT =>, QwAlarm =>)
   END_RUNG
   // the same network as SCL:
   #"AV-31.62"(LOCK := #lock,   // "Valve"
               LIOP_SEL := #Init,
               L_AUT := #Init,
               L_REMOTE := #Init,
               L_RESET := #Reset,
               L_MON := #Init,
               INSTANCE := 'AV-31.62');
END_REGION

REGION Network 134: AV-32.01
   RUNG wire#powerrail
      #"AV-32.01"(AUT_OP := wire#w1, FB_OPEN := wire#w2, FB_CLOSE := wire#w3, LOCK := #lock, ERR_EXTERN :=, LIOP_SEL := #Init, L_AUT := #Init, L_REMOTE := #Init, L_SIM :=, L_RESET := #Reset, MAN_OP :=, SIM_OP :=, L_MON := #Init, MON_T :=, MON_T_CLOSE :=, INSTANCE := 'AV-32.01', RESTART :=, VISIBILITY :=, OPdwCmd :=, QdwState =>, QwState =>, QCLOSING =>, QCLOSE =>, QOPENING =>, QOPEN =>, QCMD_OP => "AV-32.01", QMON =>, QMON_ERR =>, QMON_T =>, QMON_T_CLOSE =>, QMAN_AUT =>, QREMOTE =>, QSIM =>, QLOCK =>, QERR =>, QERR_EXT =>, QwAlarm =>)
   END_RUNG
   RUNG wire#powerrail
      Contact( "Rework_T-32_DB".Out_AV_Transfer )
      Contact( "AlwaysFALSE" )
   END_RUNG wire#w1
   RUNG wire#powerrail
      Contact( "AV-32.01" )
   END_RUNG wire#w2
   RUNG wire#powerrail
      I_Contact( "AV-32.01" )
   END_RUNG wire#w3
   // the same network as SCL:
   #"AV-32.01"(LOCK := #lock,   // "Valve"
               LIOP_SEL := #Init,
               L_AUT := #Init,
               L_REMOTE := #Init,
               L_RESET := #Reset,
               AUT_OP := "Rework_T-32_DB".Out_AV_Transfer AND "AlwaysFALSE",
               FB_OPEN := "AV-32.01",
               FB_CLOSE := NOT "AV-32.01",
               L_MON := #Init,
               INSTANCE := 'AV-32.01',
               QCMD_OP => "AV-32.01");
END_REGION

REGION Network 135: AV-32.02
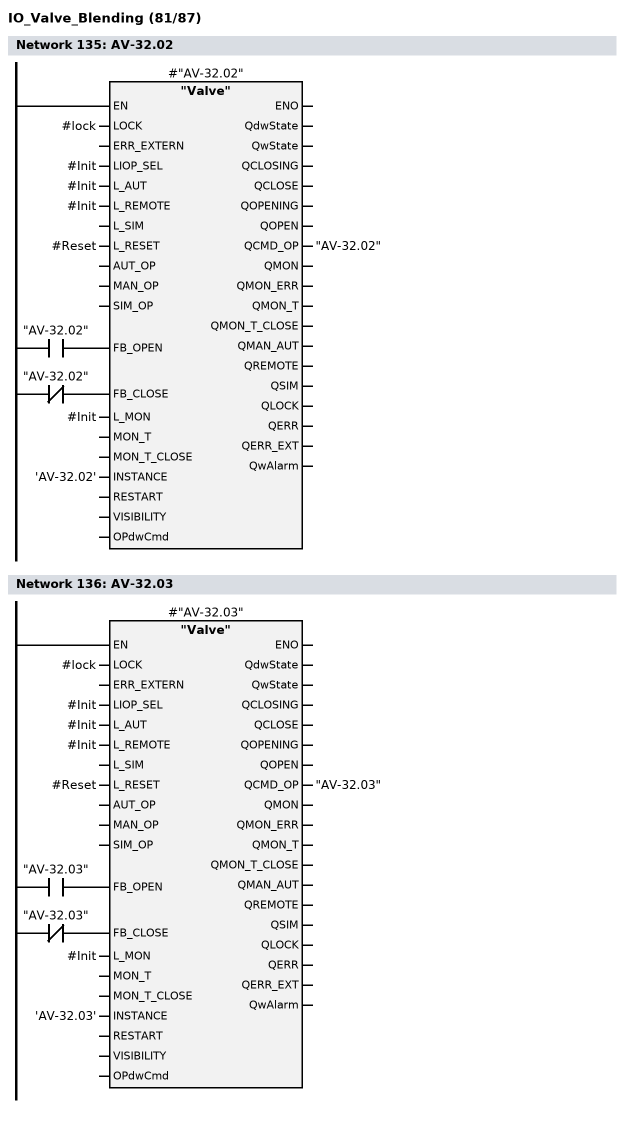
   RUNG wire#powerrail
      #"AV-32.02"(FB_OPEN := wire#w1, FB_CLOSE := wire#w2, LOCK := #lock, ERR_EXTERN :=, LIOP_SEL := #Init, L_AUT := #Init, L_REMOTE := #Init, L_SIM :=, L_RESET := #Reset, AUT_OP :=, MAN_OP :=, SIM_OP :=, L_MON := #Init, MON_T :=, MON_T_CLOSE :=, INSTANCE := 'AV-32.02', RESTART :=, VISIBILITY :=, OPdwCmd :=, QdwState =>, QwState =>, QCLOSING =>, QCLOSE =>, QOPENING =>, QOPEN =>, QCMD_OP => "AV-32.02", QMON =>, QMON_ERR =>, QMON_T =>, QMON_T_CLOSE =>, QMAN_AUT =>, QREMOTE =>, QSIM =>, QLOCK =>, QERR =>, QERR_EXT =>, QwAlarm =>)
   END_RUNG
   RUNG wire#powerrail
      Contact( "AV-32.02" )
   END_RUNG wire#w1
   RUNG wire#powerrail
      I_Contact( "AV-32.02" )
   END_RUNG wire#w2
   // the same network as SCL:
   #"AV-32.02"(LOCK := #lock,   // "Valve"
               LIOP_SEL := #Init,
               L_AUT := #Init,
               L_REMOTE := #Init,
               L_RESET := #Reset,
               FB_OPEN := "AV-32.02",
               FB_CLOSE := NOT "AV-32.02",
               L_MON := #Init,
               INSTANCE := 'AV-32.02',
               QCMD_OP => "AV-32.02");
END_REGION

REGION Network 136: AV-32.03
   RUNG wire#powerrail
      #"AV-32.03"(FB_OPEN := wire#w1, FB_CLOSE := wire#w2, LOCK := #lock, ERR_EXTERN :=, LIOP_SEL := #Init, L_AUT := #Init, L_REMOTE := #Init, L_SIM :=, L_RESET := #Reset, AUT_OP :=, MAN_OP :=, SIM_OP :=, L_MON := #Init, MON_T :=, MON_T_CLOSE :=, INSTANCE := 'AV-32.03', RESTART :=, VISIBILITY :=, OPdwCmd :=, QdwState =>, QwState =>, QCLOSING =>, QCLOSE =>, QOPENING =>, QOPEN =>, QCMD_OP => "AV-32.03", QMON =>, QMON_ERR =>, QMON_T =>, QMON_T_CLOSE =>, QMAN_AUT =>, QREMOTE =>, QSIM =>, QLOCK =>, QERR =>, QERR_EXT =>, QwAlarm =>)
   END_RUNG
   RUNG wire#powerrail
      Contact( "AV-32.03" )
   END_RUNG wire#w1
   RUNG wire#powerrail
      I_Contact( "AV-32.03" )
   END_RUNG wire#w2
   // the same network as SCL:
   #"AV-32.03"(LOCK := #lock,   // "Valve"
               LIOP_SEL := #Init,
               L_AUT := #Init,
               L_REMOTE := #Init,
               L_RESET := #Reset,
               FB_OPEN := "AV-32.03",
               FB_CLOSE := NOT "AV-32.03",
               L_MON := #Init,
               INSTANCE := 'AV-32.03',
               QCMD_OP => "AV-32.03");
END_REGION

REGION Network 137: AV-32.06
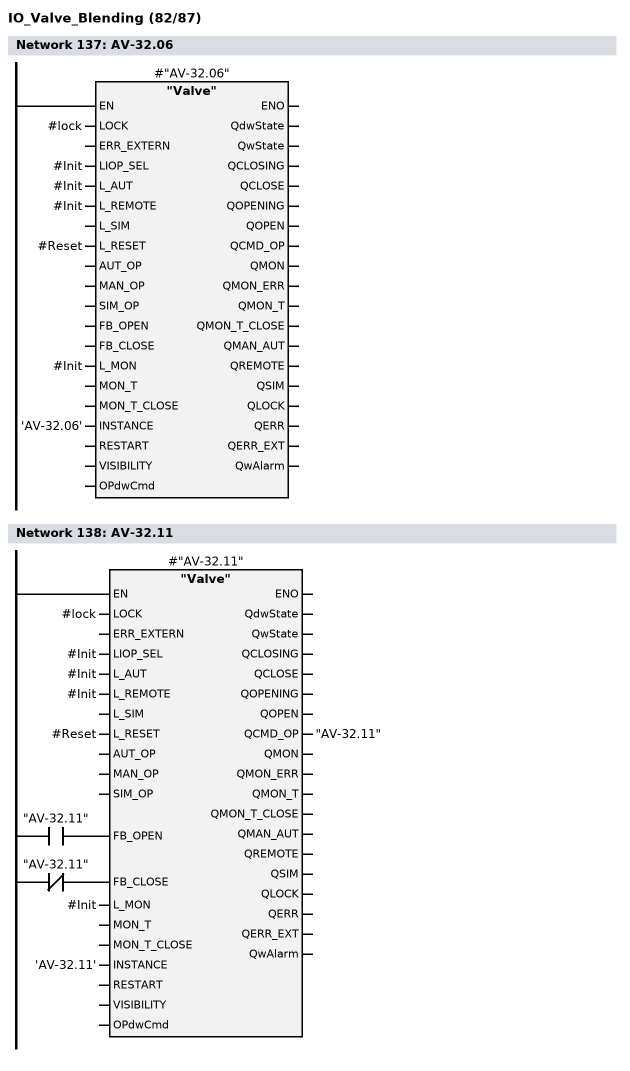
   RUNG wire#powerrail
      #"AV-32.06"(LOCK := #lock, ERR_EXTERN :=, LIOP_SEL := #Init, L_AUT := #Init, L_REMOTE := #Init, L_SIM :=, L_RESET := #Reset, AUT_OP :=, MAN_OP :=, SIM_OP :=, FB_OPEN :=, FB_CLOSE :=, L_MON := #Init, MON_T :=, MON_T_CLOSE :=, INSTANCE := 'AV-32.06', RESTART :=, VISIBILITY :=, OPdwCmd :=, QdwState =>, QwState =>, QCLOSING =>, QCLOSE =>, QOPENING =>, QOPEN =>, QCMD_OP =>, QMON =>, QMON_ERR =>, QMON_T =>, QMON_T_CLOSE =>, QMAN_AUT =>, QREMOTE =>, QSIM =>, QLOCK =>, QERR =>, QERR_EXT =>, QwAlarm =>)
   END_RUNG
   // the same network as SCL:
   #"AV-32.06"(LOCK := #lock,   // "Valve"
               LIOP_SEL := #Init,
               L_AUT := #Init,
               L_REMOTE := #Init,
               L_RESET := #Reset,
               L_MON := #Init,
               INSTANCE := 'AV-32.06');
END_REGION

REGION Network 138: AV-32.11
   RUNG wire#powerrail
      #"AV-32.11"(FB_OPEN := wire#w1, FB_CLOSE := wire#w2, LOCK := #lock, ERR_EXTERN :=, LIOP_SEL := #Init, L_AUT := #Init, L_REMOTE := #Init, L_SIM :=, L_RESET := #Reset, AUT_OP :=, MAN_OP :=, SIM_OP :=, L_MON := #Init, MON_T :=, MON_T_CLOSE :=, INSTANCE := 'AV-32.11', RESTART :=, VISIBILITY :=, OPdwCmd :=, QdwState =>, QwState =>, QCLOSING =>, QCLOSE =>, QOPENING =>, QOPEN =>, QCMD_OP => "AV-32.11", QMON =>, QMON_ERR =>, QMON_T =>, QMON_T_CLOSE =>, QMAN_AUT =>, QREMOTE =>, QSIM =>, QLOCK =>, QERR =>, QERR_EXT =>, QwAlarm =>)
   END_RUNG
   RUNG wire#powerrail
      Contact( "AV-32.11" )
   END_RUNG wire#w1
   RUNG wire#powerrail
      I_Contact( "AV-32.11" )
   END_RUNG wire#w2
   // the same network as SCL:
   #"AV-32.11"(LOCK := #lock,   // "Valve"
               LIOP_SEL := #Init,
               L_AUT := #Init,
               L_REMOTE := #Init,
               L_RESET := #Reset,
               FB_OPEN := "AV-32.11",
               FB_CLOSE := NOT "AV-32.11",
               L_MON := #Init,
               INSTANCE := 'AV-32.11',
               QCMD_OP => "AV-32.11");
END_REGION

REGION Network 139: AV-32.21
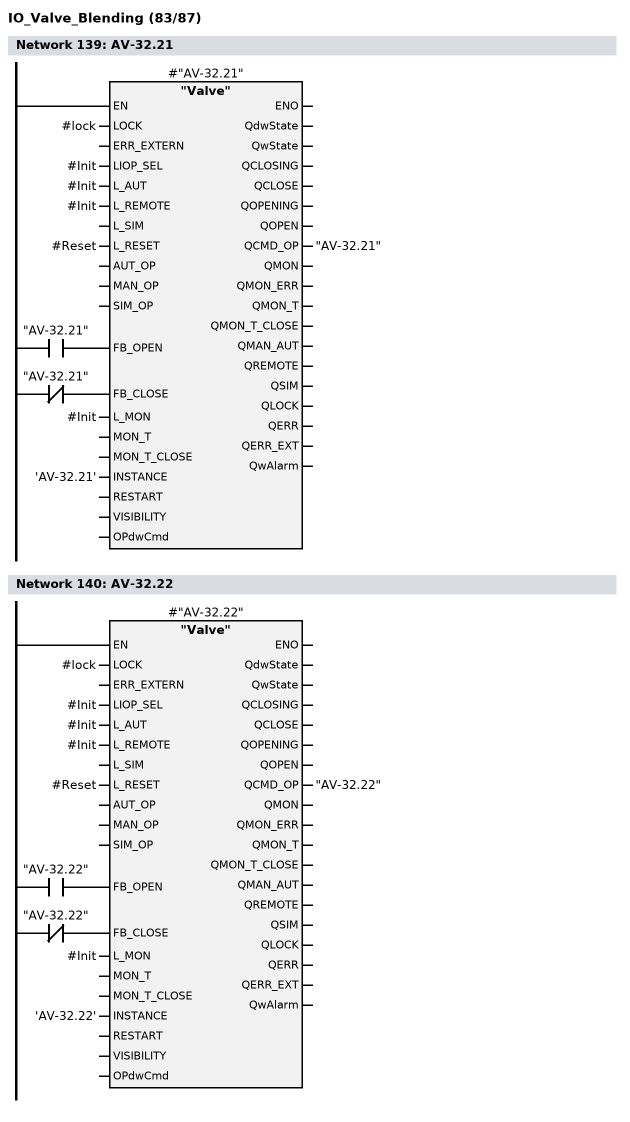
   RUNG wire#powerrail
      #"AV-32.21"(FB_OPEN := wire#w1, FB_CLOSE := wire#w2, LOCK := #lock, ERR_EXTERN :=, LIOP_SEL := #Init, L_AUT := #Init, L_REMOTE := #Init, L_SIM :=, L_RESET := #Reset, AUT_OP :=, MAN_OP :=, SIM_OP :=, L_MON := #Init, MON_T :=, MON_T_CLOSE :=, INSTANCE := 'AV-32.21', RESTART :=, VISIBILITY :=, OPdwCmd :=, QdwState =>, QwState =>, QCLOSING =>, QCLOSE =>, QOPENING =>, QOPEN =>, QCMD_OP => "AV-32.21", QMON =>, QMON_ERR =>, QMON_T =>, QMON_T_CLOSE =>, QMAN_AUT =>, QREMOTE =>, QSIM =>, QLOCK =>, QERR =>, QERR_EXT =>, QwAlarm =>)
   END_RUNG
   RUNG wire#powerrail
      Contact( "AV-32.21" )
   END_RUNG wire#w1
   RUNG wire#powerrail
      I_Contact( "AV-32.21" )
   END_RUNG wire#w2
   // the same network as SCL:
   #"AV-32.21"(LOCK := #lock,   // "Valve"
               LIOP_SEL := #Init,
               L_AUT := #Init,
               L_REMOTE := #Init,
               L_RESET := #Reset,
               FB_OPEN := "AV-32.21",
               FB_CLOSE := NOT "AV-32.21",
               L_MON := #Init,
               INSTANCE := 'AV-32.21',
               QCMD_OP => "AV-32.21");
END_REGION

REGION Network 140: AV-32.22
   RUNG wire#powerrail
      #"AV-32.22"(FB_OPEN := wire#w1, FB_CLOSE := wire#w2, LOCK := #lock, ERR_EXTERN :=, LIOP_SEL := #Init, L_AUT := #Init, L_REMOTE := #Init, L_SIM :=, L_RESET := #Reset, AUT_OP :=, MAN_OP :=, SIM_OP :=, L_MON := #Init, MON_T :=, MON_T_CLOSE :=, INSTANCE := 'AV-32.22', RESTART :=, VISIBILITY :=, OPdwCmd :=, QdwState =>, QwState =>, QCLOSING =>, QCLOSE =>, QOPENING =>, QOPEN =>, QCMD_OP => "AV-32.22", QMON =>, QMON_ERR =>, QMON_T =>, QMON_T_CLOSE =>, QMAN_AUT =>, QREMOTE =>, QSIM =>, QLOCK =>, QERR =>, QERR_EXT =>, QwAlarm =>)
   END_RUNG
   RUNG wire#powerrail
      Contact( "AV-32.22" )
   END_RUNG wire#w1
   RUNG wire#powerrail
      I_Contact( "AV-32.22" )
   END_RUNG wire#w2
   // the same network as SCL:
   #"AV-32.22"(LOCK := #lock,   // "Valve"
               LIOP_SEL := #Init,
               L_AUT := #Init,
               L_REMOTE := #Init,
               L_RESET := #Reset,
               FB_OPEN := "AV-32.22",
               FB_CLOSE := NOT "AV-32.22",
               L_MON := #Init,
               INSTANCE := 'AV-32.22',
               QCMD_OP => "AV-32.22");
END_REGION

REGION Network 141: AV-20.42
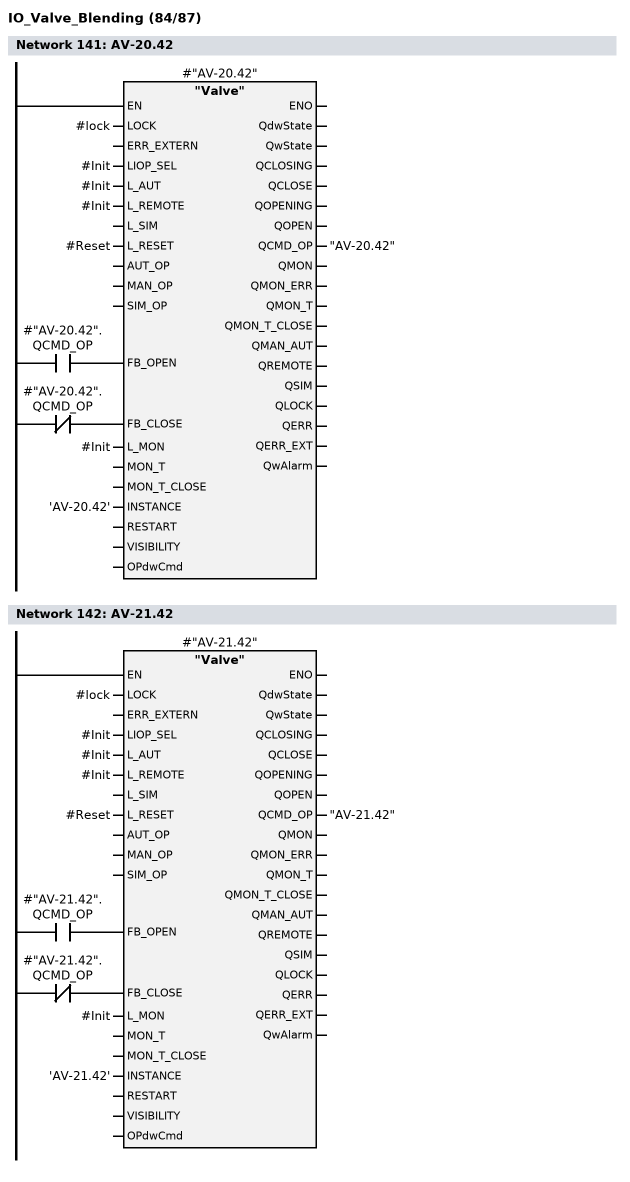
   RUNG wire#powerrail
      #"AV-20.42"(FB_OPEN := wire#w1, FB_CLOSE := wire#w2, LOCK := #lock, ERR_EXTERN :=, LIOP_SEL := #Init, L_AUT := #Init, L_REMOTE := #Init, L_SIM :=, L_RESET := #Reset, AUT_OP :=, MAN_OP :=, SIM_OP :=, L_MON := #Init, MON_T :=, MON_T_CLOSE :=, INSTANCE := 'AV-20.42', RESTART :=, VISIBILITY :=, OPdwCmd :=, QdwState =>, QwState =>, QCLOSING =>, QCLOSE =>, QOPENING =>, QOPEN =>, QCMD_OP => "AV-20.42", QMON =>, QMON_ERR =>, QMON_T =>, QMON_T_CLOSE =>, QMAN_AUT =>, QREMOTE =>, QSIM =>, QLOCK =>, QERR =>, QERR_EXT =>, QwAlarm =>)
   END_RUNG
   RUNG wire#powerrail
      Contact( #"AV-20.42".QCMD_OP )
   END_RUNG wire#w1
   RUNG wire#powerrail
      I_Contact( #"AV-20.42".QCMD_OP )
   END_RUNG wire#w2
   // the same network as SCL:
   #"AV-20.42"(LOCK := #lock,   // "Valve"
               LIOP_SEL := #Init,
               L_AUT := #Init,
               L_REMOTE := #Init,
               L_RESET := #Reset,
               FB_OPEN := #"AV-20.42".QCMD_OP,
               FB_CLOSE := NOT #"AV-20.42".QCMD_OP,
               L_MON := #Init,
               INSTANCE := 'AV-20.42',
               QCMD_OP => "AV-20.42");
END_REGION

REGION Network 142: AV-21.42
   RUNG wire#powerrail
      #"AV-21.42"(FB_OPEN := wire#w1, FB_CLOSE := wire#w2, LOCK := #lock, ERR_EXTERN :=, LIOP_SEL := #Init, L_AUT := #Init, L_REMOTE := #Init, L_SIM :=, L_RESET := #Reset, AUT_OP :=, MAN_OP :=, SIM_OP :=, L_MON := #Init, MON_T :=, MON_T_CLOSE :=, INSTANCE := 'AV-21.42', RESTART :=, VISIBILITY :=, OPdwCmd :=, QdwState =>, QwState =>, QCLOSING =>, QCLOSE =>, QOPENING =>, QOPEN =>, QCMD_OP => "AV-21.42", QMON =>, QMON_ERR =>, QMON_T =>, QMON_T_CLOSE =>, QMAN_AUT =>, QREMOTE =>, QSIM =>, QLOCK =>, QERR =>, QERR_EXT =>, QwAlarm =>)
   END_RUNG
   RUNG wire#powerrail
      Contact( #"AV-21.42".QCMD_OP )
   END_RUNG wire#w1
   RUNG wire#powerrail
      I_Contact( #"AV-21.42".QCMD_OP )
   END_RUNG wire#w2
   // the same network as SCL:
   #"AV-21.42"(LOCK := #lock,   // "Valve"
               LIOP_SEL := #Init,
               L_AUT := #Init,
               L_REMOTE := #Init,
               L_RESET := #Reset,
               FB_OPEN := #"AV-21.42".QCMD_OP,
               FB_CLOSE := NOT #"AV-21.42".QCMD_OP,
               L_MON := #Init,
               INSTANCE := 'AV-21.42',
               QCMD_OP => "AV-21.42");
END_REGION

REGION Network 143: AV-22.04
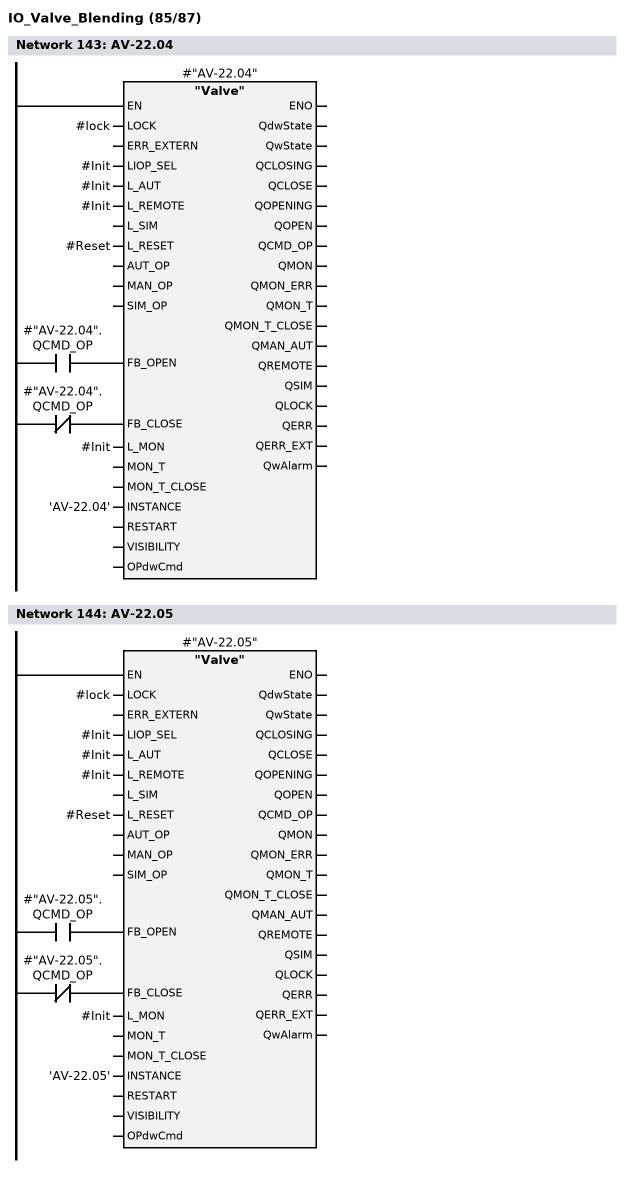
   RUNG wire#powerrail
      #"AV-22.04"(FB_OPEN := wire#w1, FB_CLOSE := wire#w2, LOCK := #lock, ERR_EXTERN :=, LIOP_SEL := #Init, L_AUT := #Init, L_REMOTE := #Init, L_SIM :=, L_RESET := #Reset, AUT_OP :=, MAN_OP :=, SIM_OP :=, L_MON := #Init, MON_T :=, MON_T_CLOSE :=, INSTANCE := 'AV-22.04', RESTART :=, VISIBILITY :=, OPdwCmd :=, QdwState =>, QwState =>, QCLOSING =>, QCLOSE =>, QOPENING =>, QOPEN =>, QCMD_OP =>, QMON =>, QMON_ERR =>, QMON_T =>, QMON_T_CLOSE =>, QMAN_AUT =>, QREMOTE =>, QSIM =>, QLOCK =>, QERR =>, QERR_EXT =>, QwAlarm =>)
   END_RUNG
   RUNG wire#powerrail
      Contact( #"AV-22.04".QCMD_OP )
   END_RUNG wire#w1
   RUNG wire#powerrail
      I_Contact( #"AV-22.04".QCMD_OP )
   END_RUNG wire#w2
   // the same network as SCL:
   #"AV-22.04"(LOCK := #lock,   // "Valve"
               LIOP_SEL := #Init,
               L_AUT := #Init,
               L_REMOTE := #Init,
               L_RESET := #Reset,
               FB_OPEN := #"AV-22.04".QCMD_OP,
               FB_CLOSE := NOT #"AV-22.04".QCMD_OP,
               L_MON := #Init,
               INSTANCE := 'AV-22.04');
END_REGION

REGION Network 144: AV-22.05
   RUNG wire#powerrail
      #"AV-22.05"(FB_OPEN := wire#w1, FB_CLOSE := wire#w2, LOCK := #lock, ERR_EXTERN :=, LIOP_SEL := #Init, L_AUT := #Init, L_REMOTE := #Init, L_SIM :=, L_RESET := #Reset, AUT_OP :=, MAN_OP :=, SIM_OP :=, L_MON := #Init, MON_T :=, MON_T_CLOSE :=, INSTANCE := 'AV-22.05', RESTART :=, VISIBILITY :=, OPdwCmd :=, QdwState =>, QwState =>, QCLOSING =>, QCLOSE =>, QOPENING =>, QOPEN =>, QCMD_OP =>, QMON =>, QMON_ERR =>, QMON_T =>, QMON_T_CLOSE =>, QMAN_AUT =>, QREMOTE =>, QSIM =>, QLOCK =>, QERR =>, QERR_EXT =>, QwAlarm =>)
   END_RUNG
   RUNG wire#powerrail
      Contact( #"AV-22.05".QCMD_OP )
   END_RUNG wire#w1
   RUNG wire#powerrail
      I_Contact( #"AV-22.05".QCMD_OP )
   END_RUNG wire#w2
   // the same network as SCL:
   #"AV-22.05"(LOCK := #lock,   // "Valve"
               LIOP_SEL := #Init,
               L_AUT := #Init,
               L_REMOTE := #Init,
               L_RESET := #Reset,
               FB_OPEN := #"AV-22.05".QCMD_OP,
               FB_CLOSE := NOT #"AV-22.05".QCMD_OP,
               L_MON := #Init,
               INSTANCE := 'AV-22.05');
END_REGION

REGION Network 145: AV-30.42
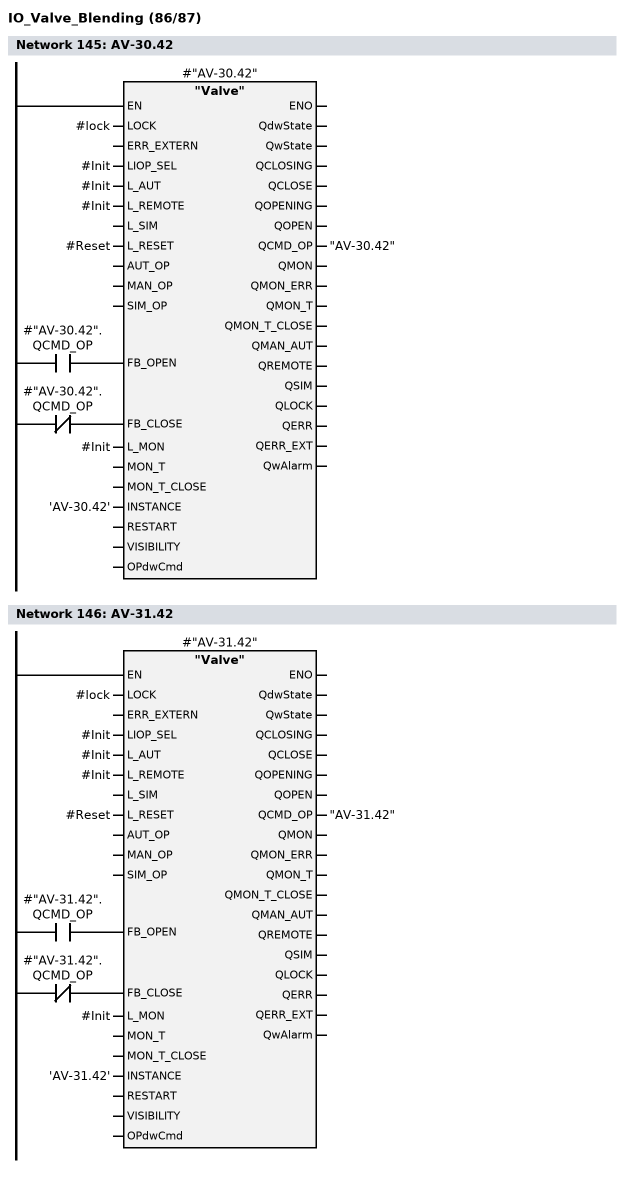
   RUNG wire#powerrail
      #"AV-30.42"(FB_OPEN := wire#w1, FB_CLOSE := wire#w2, LOCK := #lock, ERR_EXTERN :=, LIOP_SEL := #Init, L_AUT := #Init, L_REMOTE := #Init, L_SIM :=, L_RESET := #Reset, AUT_OP :=, MAN_OP :=, SIM_OP :=, L_MON := #Init, MON_T :=, MON_T_CLOSE :=, INSTANCE := 'AV-30.42', RESTART :=, VISIBILITY :=, OPdwCmd :=, QdwState =>, QwState =>, QCLOSING =>, QCLOSE =>, QOPENING =>, QOPEN =>, QCMD_OP => "AV-30.42", QMON =>, QMON_ERR =>, QMON_T =>, QMON_T_CLOSE =>, QMAN_AUT =>, QREMOTE =>, QSIM =>, QLOCK =>, QERR =>, QERR_EXT =>, QwAlarm =>)
   END_RUNG
   RUNG wire#powerrail
      Contact( #"AV-30.42".QCMD_OP )
   END_RUNG wire#w1
   RUNG wire#powerrail
      I_Contact( #"AV-30.42".QCMD_OP )
   END_RUNG wire#w2
   // the same network as SCL:
   #"AV-30.42"(LOCK := #lock,   // "Valve"
               LIOP_SEL := #Init,
               L_AUT := #Init,
               L_REMOTE := #Init,
               L_RESET := #Reset,
               FB_OPEN := #"AV-30.42".QCMD_OP,
               FB_CLOSE := NOT #"AV-30.42".QCMD_OP,
               L_MON := #Init,
               INSTANCE := 'AV-30.42',
               QCMD_OP => "AV-30.42");
END_REGION

REGION Network 146: AV-31.42
   RUNG wire#powerrail
      #"AV-31.42"(FB_OPEN := wire#w1, FB_CLOSE := wire#w2, LOCK := #lock, ERR_EXTERN :=, LIOP_SEL := #Init, L_AUT := #Init, L_REMOTE := #Init, L_SIM :=, L_RESET := #Reset, AUT_OP :=, MAN_OP :=, SIM_OP :=, L_MON := #Init, MON_T :=, MON_T_CLOSE :=, INSTANCE := 'AV-31.42', RESTART :=, VISIBILITY :=, OPdwCmd :=, QdwState =>, QwState =>, QCLOSING =>, QCLOSE =>, QOPENING =>, QOPEN =>, QCMD_OP => "AV-31.42", QMON =>, QMON_ERR =>, QMON_T =>, QMON_T_CLOSE =>, QMAN_AUT =>, QREMOTE =>, QSIM =>, QLOCK =>, QERR =>, QERR_EXT =>, QwAlarm =>)
   END_RUNG
   RUNG wire#powerrail
      Contact( #"AV-31.42".QCMD_OP )
   END_RUNG wire#w1
   RUNG wire#powerrail
      I_Contact( #"AV-31.42".QCMD_OP )
   END_RUNG wire#w2
   // the same network as SCL:
   #"AV-31.42"(LOCK := #lock,   // "Valve"
               LIOP_SEL := #Init,
               L_AUT := #Init,
               L_REMOTE := #Init,
               L_RESET := #Reset,
               FB_OPEN := #"AV-31.42".QCMD_OP,
               FB_CLOSE := NOT #"AV-31.42".QCMD_OP,
               L_MON := #Init,
               INSTANCE := 'AV-31.42',
               QCMD_OP => "AV-31.42");
END_REGION

REGION Network 147: AV-32.04
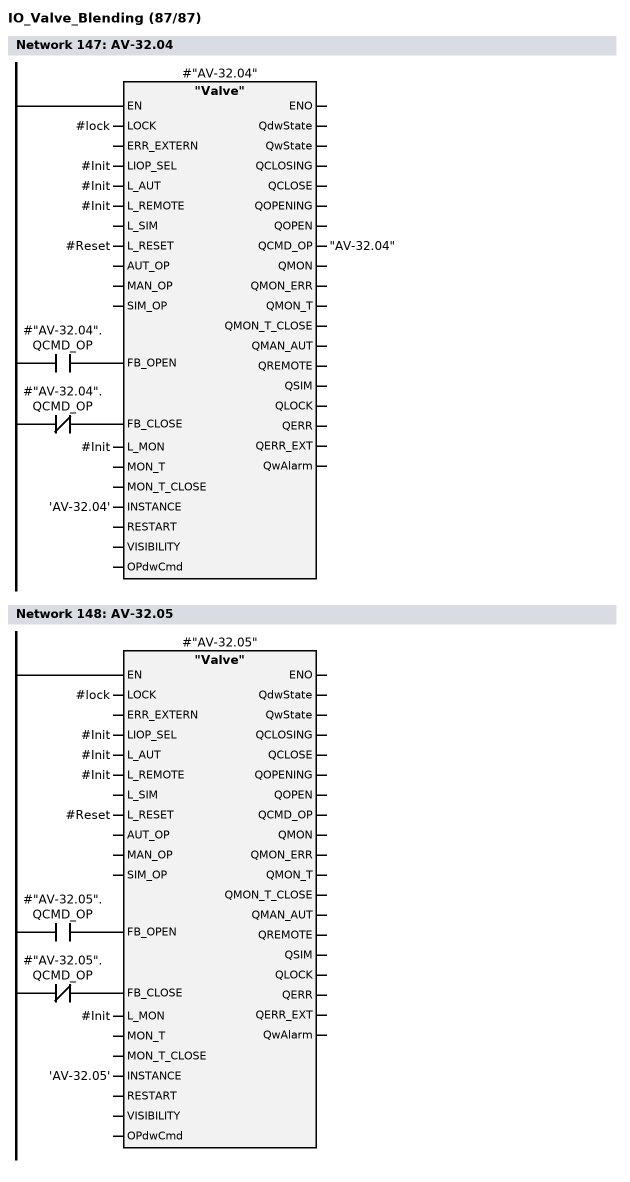
   RUNG wire#powerrail
      #"AV-32.04"(FB_OPEN := wire#w1, FB_CLOSE := wire#w2, LOCK := #lock, ERR_EXTERN :=, LIOP_SEL := #Init, L_AUT := #Init, L_REMOTE := #Init, L_SIM :=, L_RESET := #Reset, AUT_OP :=, MAN_OP :=, SIM_OP :=, L_MON := #Init, MON_T :=, MON_T_CLOSE :=, INSTANCE := 'AV-32.04', RESTART :=, VISIBILITY :=, OPdwCmd :=, QdwState =>, QwState =>, QCLOSING =>, QCLOSE =>, QOPENING =>, QOPEN =>, QCMD_OP => "AV-32.04", QMON =>, QMON_ERR =>, QMON_T =>, QMON_T_CLOSE =>, QMAN_AUT =>, QREMOTE =>, QSIM =>, QLOCK =>, QERR =>, QERR_EXT =>, QwAlarm =>)
   END_RUNG
   RUNG wire#powerrail
      Contact( #"AV-32.04".QCMD_OP )
   END_RUNG wire#w1
   RUNG wire#powerrail
      I_Contact( #"AV-32.04".QCMD_OP )
   END_RUNG wire#w2
   // the same network as SCL:
   #"AV-32.04"(LOCK := #lock,   // "Valve"
               LIOP_SEL := #Init,
               L_AUT := #Init,
               L_REMOTE := #Init,
               L_RESET := #Reset,
               FB_OPEN := #"AV-32.04".QCMD_OP,
               FB_CLOSE := NOT #"AV-32.04".QCMD_OP,
               L_MON := #Init,
               INSTANCE := 'AV-32.04',
               QCMD_OP => "AV-32.04");
END_REGION

REGION Network 148: AV-32.05
   RUNG wire#powerrail
      #"AV-32.05"(FB_OPEN := wire#w1, FB_CLOSE := wire#w2, LOCK := #lock, ERR_EXTERN :=, LIOP_SEL := #Init, L_AUT := #Init, L_REMOTE := #Init, L_SIM :=, L_RESET := #Reset, AUT_OP :=, MAN_OP :=, SIM_OP :=, L_MON := #Init, MON_T :=, MON_T_CLOSE :=, INSTANCE := 'AV-32.05', RESTART :=, VISIBILITY :=, OPdwCmd :=, QdwState =>, QwState =>, QCLOSING =>, QCLOSE =>, QOPENING =>, QOPEN =>, QCMD_OP =>, QMON =>, QMON_ERR =>, QMON_T =>, QMON_T_CLOSE =>, QMAN_AUT =>, QREMOTE =>, QSIM =>, QLOCK =>, QERR =>, QERR_EXT =>, QwAlarm =>)
   END_RUNG
   RUNG wire#powerrail
      Contact( #"AV-32.05".QCMD_OP )
   END_RUNG wire#w1
   RUNG wire#powerrail
      I_Contact( #"AV-32.05".QCMD_OP )
   END_RUNG wire#w2
   // the same network as SCL:
   #"AV-32.05"(LOCK := #lock,   // "Valve"
               LIOP_SEL := #Init,
               L_AUT := #Init,
               L_REMOTE := #Init,
               L_RESET := #Reset,
               FB_OPEN := #"AV-32.05".QCMD_OP,
               FB_CLOSE := NOT #"AV-32.05".QCMD_OP,
               L_MON := #Init,
               INSTANCE := 'AV-32.05');
END_REGION
END_FUNCTION_BLOCK

FUNCTION_BLOCK "IO Valve T01 HWT"   // FB301, LAD
{ S7_Optimized_Access := 'FALSE' }
VERSION : 0.1
// stored: AutoNumber false, IsIECCheckEnabled false, SetENOAutomatically false, UDAEnableTagReadback false
   VAR_INPUT
      lock : Bool;
      Init : Bool;
      Reset : Bool;
   END_VAR
   VAR
      "AV-01.01" { S7_SetPoint := 'True'} : "Valve";   // AUTO BUTTERFLY VALVE INLET HOT WATER CIRC. TO HOT WATER TANK T-01.00
      "AV-01.02" { S7_SetPoint := 'True'} : "Valve";   // AUTO BUTTERFLY VALVE INLET PROCESS WATER TO HOT WATER TANK T-01.00
      "AV-01.03" { S7_SetPoint := 'True'} : "Valve";   // AUTO BUTTERFLY VALVE CIP RETURN LINE 1
      "AV-01.04" { S7_SetPoint := 'True'} : "Valve";   // AUTO BUTTERFLY VALVE CIP SUPPLY HOT WATER TANK T-01.00
      "AV-01.05" { S7_SetPoint := 'True'} : "Valve";
      "AV-01.06" { S7_SetPoint := 'True'} : "Valve";
      "AV-01.07" { S7_SetPoint := 'True'} : "Valve";
      "AV-01.08" { S7_SetPoint := 'True'} : "Valve";
      "AV-01.09" { S7_SetPoint := 'True'} : "Valve";
      "AV-01.10" { S7_SetPoint := 'True'} : "Valve";   // AUTO ANGLE SEAT VALVE STEAM SUPPLY
      "AV-01.11" { S7_SetPoint := 'True'} : "Valve";
      "AV-01.12" { S7_SetPoint := 'True'} : "Valve";
      "AV-01.13" { S7_SetPoint := 'True'} : "Valve";
      "AV-01.14" { S7_SetPoint := 'True'} : "Valve";
      "AV-01.15" { S7_SetPoint := 'True'} : "Valve";
      "CV-01.01" { S7_SetPoint := 'True'} : "Valve";   // CONTROL VALVE STEAM FOR PHE PROCESS PHE-01.01
   END_VAR
BEGIN

REGION Network 1: AV-01.01
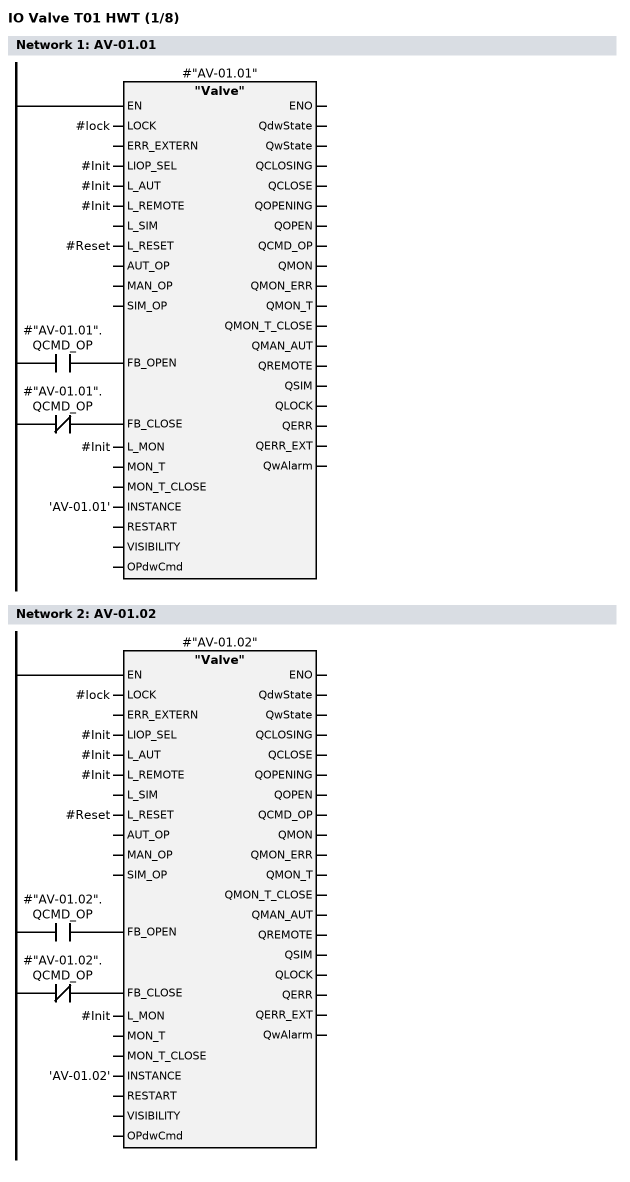
   RUNG wire#powerrail
      #"AV-01.01"(FB_OPEN := wire#w1, FB_CLOSE := wire#w2, LOCK := #lock, ERR_EXTERN :=, LIOP_SEL := #Init, L_AUT := #Init, L_REMOTE := #Init, L_SIM :=, L_RESET := #Reset, AUT_OP :=, MAN_OP :=, SIM_OP :=, L_MON := #Init, MON_T :=, MON_T_CLOSE :=, INSTANCE := 'AV-01.01', RESTART :=, VISIBILITY :=, OPdwCmd :=, QdwState =>, QwState =>, QCLOSING =>, QCLOSE =>, QOPENING =>, QOPEN =>, QCMD_OP =>, QMON =>, QMON_ERR =>, QMON_T =>, QMON_T_CLOSE =>, QMAN_AUT =>, QREMOTE =>, QSIM =>, QLOCK =>, QERR =>, QERR_EXT =>, QwAlarm =>)
   END_RUNG
   RUNG wire#powerrail
      Contact( #"AV-01.01".QCMD_OP )
   END_RUNG wire#w1
   RUNG wire#powerrail
      I_Contact( #"AV-01.01".QCMD_OP )
   END_RUNG wire#w2
   // the same network as SCL:
   #"AV-01.01"(LOCK := #lock,   // "Valve"
               LIOP_SEL := #Init,
               L_AUT := #Init,
               L_REMOTE := #Init,
               L_RESET := #Reset,
               FB_OPEN := #"AV-01.01".QCMD_OP,
               FB_CLOSE := NOT #"AV-01.01".QCMD_OP,
               L_MON := #Init,
               INSTANCE := 'AV-01.01');
END_REGION

REGION Network 2: AV-01.02
   RUNG wire#powerrail
      #"AV-01.02"(FB_OPEN := wire#w1, FB_CLOSE := wire#w2, LOCK := #lock, ERR_EXTERN :=, LIOP_SEL := #Init, L_AUT := #Init, L_REMOTE := #Init, L_SIM :=, L_RESET := #Reset, AUT_OP :=, MAN_OP :=, SIM_OP :=, L_MON := #Init, MON_T :=, MON_T_CLOSE :=, INSTANCE := 'AV-01.02', RESTART :=, VISIBILITY :=, OPdwCmd :=, QdwState =>, QwState =>, QCLOSING =>, QCLOSE =>, QOPENING =>, QOPEN =>, QCMD_OP =>, QMON =>, QMON_ERR =>, QMON_T =>, QMON_T_CLOSE =>, QMAN_AUT =>, QREMOTE =>, QSIM =>, QLOCK =>, QERR =>, QERR_EXT =>, QwAlarm =>)
   END_RUNG
   RUNG wire#powerrail
      Contact( #"AV-01.02".QCMD_OP )
   END_RUNG wire#w1
   RUNG wire#powerrail
      I_Contact( #"AV-01.02".QCMD_OP )
   END_RUNG wire#w2
   // the same network as SCL:
   #"AV-01.02"(LOCK := #lock,   // "Valve"
               LIOP_SEL := #Init,
               L_AUT := #Init,
               L_REMOTE := #Init,
               L_RESET := #Reset,
               FB_OPEN := #"AV-01.02".QCMD_OP,
               FB_CLOSE := NOT #"AV-01.02".QCMD_OP,
               L_MON := #Init,
               INSTANCE := 'AV-01.02');
END_REGION

REGION Network 3: AV-01.03
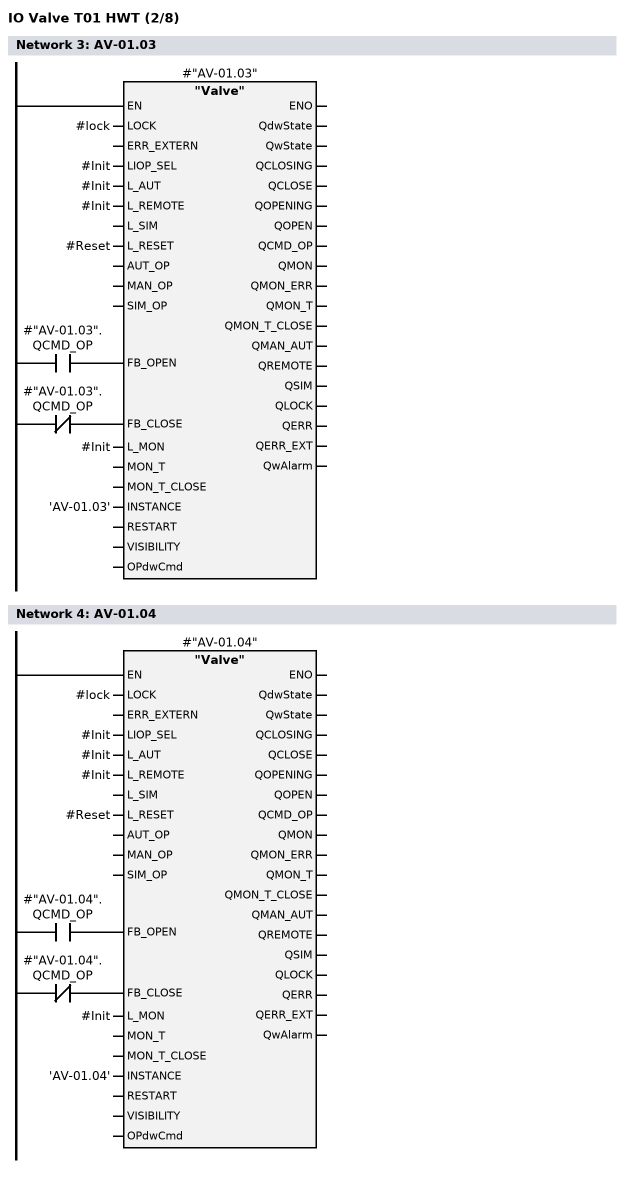
   RUNG wire#powerrail
      #"AV-01.03"(FB_OPEN := wire#w1, FB_CLOSE := wire#w2, LOCK := #lock, ERR_EXTERN :=, LIOP_SEL := #Init, L_AUT := #Init, L_REMOTE := #Init, L_SIM :=, L_RESET := #Reset, AUT_OP :=, MAN_OP :=, SIM_OP :=, L_MON := #Init, MON_T :=, MON_T_CLOSE :=, INSTANCE := 'AV-01.03', RESTART :=, VISIBILITY :=, OPdwCmd :=, QdwState =>, QwState =>, QCLOSING =>, QCLOSE =>, QOPENING =>, QOPEN =>, QCMD_OP =>, QMON =>, QMON_ERR =>, QMON_T =>, QMON_T_CLOSE =>, QMAN_AUT =>, QREMOTE =>, QSIM =>, QLOCK =>, QERR =>, QERR_EXT =>, QwAlarm =>)
   END_RUNG
   RUNG wire#powerrail
      Contact( #"AV-01.03".QCMD_OP )
   END_RUNG wire#w1
   RUNG wire#powerrail
      I_Contact( #"AV-01.03".QCMD_OP )
   END_RUNG wire#w2
   // the same network as SCL:
   #"AV-01.03"(LOCK := #lock,   // "Valve"
               LIOP_SEL := #Init,
               L_AUT := #Init,
               L_REMOTE := #Init,
               L_RESET := #Reset,
               FB_OPEN := #"AV-01.03".QCMD_OP,
               FB_CLOSE := NOT #"AV-01.03".QCMD_OP,
               L_MON := #Init,
               INSTANCE := 'AV-01.03');
END_REGION

REGION Network 4: AV-01.04
   RUNG wire#powerrail
      #"AV-01.04"(FB_OPEN := wire#w1, FB_CLOSE := wire#w2, LOCK := #lock, ERR_EXTERN :=, LIOP_SEL := #Init, L_AUT := #Init, L_REMOTE := #Init, L_SIM :=, L_RESET := #Reset, AUT_OP :=, MAN_OP :=, SIM_OP :=, L_MON := #Init, MON_T :=, MON_T_CLOSE :=, INSTANCE := 'AV-01.04', RESTART :=, VISIBILITY :=, OPdwCmd :=, QdwState =>, QwState =>, QCLOSING =>, QCLOSE =>, QOPENING =>, QOPEN =>, QCMD_OP =>, QMON =>, QMON_ERR =>, QMON_T =>, QMON_T_CLOSE =>, QMAN_AUT =>, QREMOTE =>, QSIM =>, QLOCK =>, QERR =>, QERR_EXT =>, QwAlarm =>)
   END_RUNG
   RUNG wire#powerrail
      Contact( #"AV-01.04".QCMD_OP )
   END_RUNG wire#w1
   RUNG wire#powerrail
      I_Contact( #"AV-01.04".QCMD_OP )
   END_RUNG wire#w2
   // the same network as SCL:
   #"AV-01.04"(LOCK := #lock,   // "Valve"
               LIOP_SEL := #Init,
               L_AUT := #Init,
               L_REMOTE := #Init,
               L_RESET := #Reset,
               FB_OPEN := #"AV-01.04".QCMD_OP,
               FB_CLOSE := NOT #"AV-01.04".QCMD_OP,
               L_MON := #Init,
               INSTANCE := 'AV-01.04');
END_REGION

REGION Network 5: AV-01.05
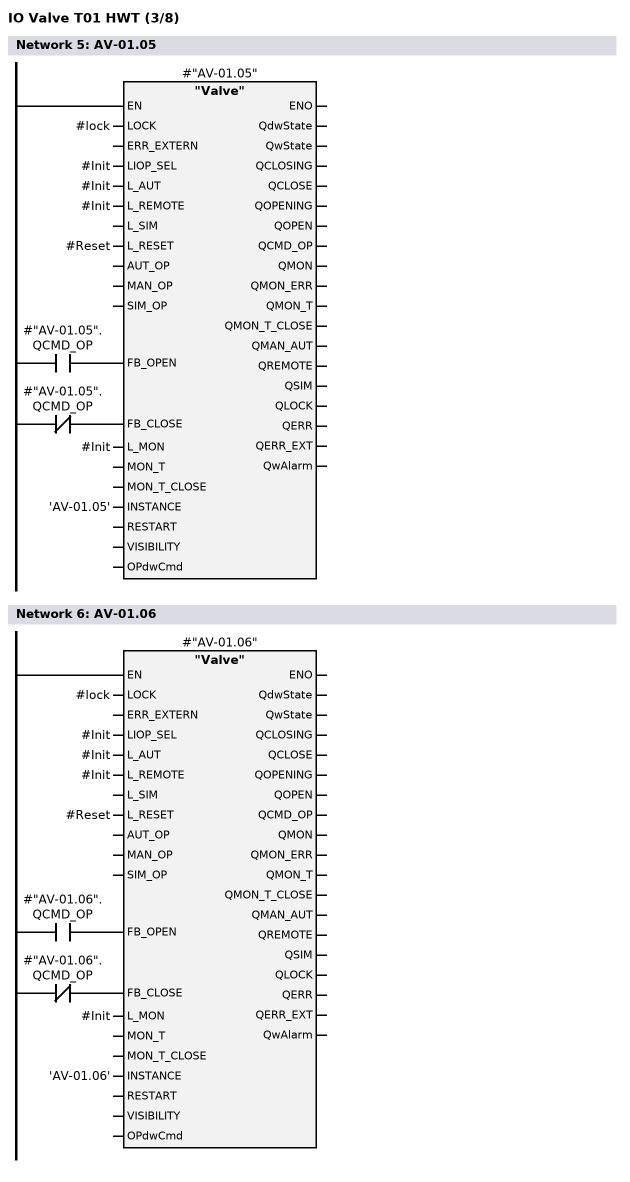
   RUNG wire#powerrail
      #"AV-01.05"(FB_OPEN := wire#w1, FB_CLOSE := wire#w2, LOCK := #lock, ERR_EXTERN :=, LIOP_SEL := #Init, L_AUT := #Init, L_REMOTE := #Init, L_SIM :=, L_RESET := #Reset, AUT_OP :=, MAN_OP :=, SIM_OP :=, L_MON := #Init, MON_T :=, MON_T_CLOSE :=, INSTANCE := 'AV-01.05', RESTART :=, VISIBILITY :=, OPdwCmd :=, QdwState =>, QwState =>, QCLOSING =>, QCLOSE =>, QOPENING =>, QOPEN =>, QCMD_OP =>, QMON =>, QMON_ERR =>, QMON_T =>, QMON_T_CLOSE =>, QMAN_AUT =>, QREMOTE =>, QSIM =>, QLOCK =>, QERR =>, QERR_EXT =>, QwAlarm =>)
   END_RUNG
   RUNG wire#powerrail
      Contact( #"AV-01.05".QCMD_OP )
   END_RUNG wire#w1
   RUNG wire#powerrail
      I_Contact( #"AV-01.05".QCMD_OP )
   END_RUNG wire#w2
   // the same network as SCL:
   #"AV-01.05"(LOCK := #lock,   // "Valve"
               LIOP_SEL := #Init,
               L_AUT := #Init,
               L_REMOTE := #Init,
               L_RESET := #Reset,
               FB_OPEN := #"AV-01.05".QCMD_OP,
               FB_CLOSE := NOT #"AV-01.05".QCMD_OP,
               L_MON := #Init,
               INSTANCE := 'AV-01.05');
END_REGION

REGION Network 6: AV-01.06
   RUNG wire#powerrail
      #"AV-01.06"(FB_OPEN := wire#w1, FB_CLOSE := wire#w2, LOCK := #lock, ERR_EXTERN :=, LIOP_SEL := #Init, L_AUT := #Init, L_REMOTE := #Init, L_SIM :=, L_RESET := #Reset, AUT_OP :=, MAN_OP :=, SIM_OP :=, L_MON := #Init, MON_T :=, MON_T_CLOSE :=, INSTANCE := 'AV-01.06', RESTART :=, VISIBILITY :=, OPdwCmd :=, QdwState =>, QwState =>, QCLOSING =>, QCLOSE =>, QOPENING =>, QOPEN =>, QCMD_OP =>, QMON =>, QMON_ERR =>, QMON_T =>, QMON_T_CLOSE =>, QMAN_AUT =>, QREMOTE =>, QSIM =>, QLOCK =>, QERR =>, QERR_EXT =>, QwAlarm =>)
   END_RUNG
   RUNG wire#powerrail
      Contact( #"AV-01.06".QCMD_OP )
   END_RUNG wire#w1
   RUNG wire#powerrail
      I_Contact( #"AV-01.06".QCMD_OP )
   END_RUNG wire#w2
   // the same network as SCL:
   #"AV-01.06"(LOCK := #lock,   // "Valve"
               LIOP_SEL := #Init,
               L_AUT := #Init,
               L_REMOTE := #Init,
               L_RESET := #Reset,
               FB_OPEN := #"AV-01.06".QCMD_OP,
               FB_CLOSE := NOT #"AV-01.06".QCMD_OP,
               L_MON := #Init,
               INSTANCE := 'AV-01.06');
END_REGION

REGION Network 7: AV-01.07
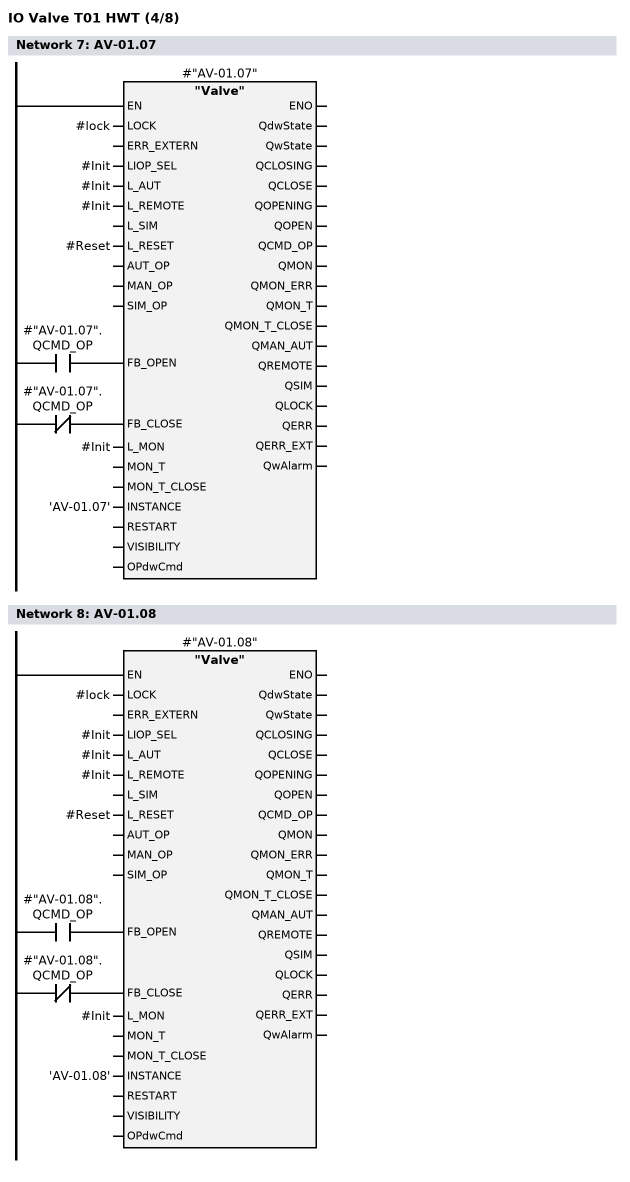
   RUNG wire#powerrail
      #"AV-01.07"(FB_OPEN := wire#w1, FB_CLOSE := wire#w2, LOCK := #lock, ERR_EXTERN :=, LIOP_SEL := #Init, L_AUT := #Init, L_REMOTE := #Init, L_SIM :=, L_RESET := #Reset, AUT_OP :=, MAN_OP :=, SIM_OP :=, L_MON := #Init, MON_T :=, MON_T_CLOSE :=, INSTANCE := 'AV-01.07', RESTART :=, VISIBILITY :=, OPdwCmd :=, QdwState =>, QwState =>, QCLOSING =>, QCLOSE =>, QOPENING =>, QOPEN =>, QCMD_OP =>, QMON =>, QMON_ERR =>, QMON_T =>, QMON_T_CLOSE =>, QMAN_AUT =>, QREMOTE =>, QSIM =>, QLOCK =>, QERR =>, QERR_EXT =>, QwAlarm =>)
   END_RUNG
   RUNG wire#powerrail
      Contact( #"AV-01.07".QCMD_OP )
   END_RUNG wire#w1
   RUNG wire#powerrail
      I_Contact( #"AV-01.07".QCMD_OP )
   END_RUNG wire#w2
   // the same network as SCL:
   #"AV-01.07"(LOCK := #lock,   // "Valve"
               LIOP_SEL := #Init,
               L_AUT := #Init,
               L_REMOTE := #Init,
               L_RESET := #Reset,
               FB_OPEN := #"AV-01.07".QCMD_OP,
               FB_CLOSE := NOT #"AV-01.07".QCMD_OP,
               L_MON := #Init,
               INSTANCE := 'AV-01.07');
END_REGION

REGION Network 8: AV-01.08
   RUNG wire#powerrail
      #"AV-01.08"(FB_OPEN := wire#w1, FB_CLOSE := wire#w2, LOCK := #lock, ERR_EXTERN :=, LIOP_SEL := #Init, L_AUT := #Init, L_REMOTE := #Init, L_SIM :=, L_RESET := #Reset, AUT_OP :=, MAN_OP :=, SIM_OP :=, L_MON := #Init, MON_T :=, MON_T_CLOSE :=, INSTANCE := 'AV-01.08', RESTART :=, VISIBILITY :=, OPdwCmd :=, QdwState =>, QwState =>, QCLOSING =>, QCLOSE =>, QOPENING =>, QOPEN =>, QCMD_OP =>, QMON =>, QMON_ERR =>, QMON_T =>, QMON_T_CLOSE =>, QMAN_AUT =>, QREMOTE =>, QSIM =>, QLOCK =>, QERR =>, QERR_EXT =>, QwAlarm =>)
   END_RUNG
   RUNG wire#powerrail
      Contact( #"AV-01.08".QCMD_OP )
   END_RUNG wire#w1
   RUNG wire#powerrail
      I_Contact( #"AV-01.08".QCMD_OP )
   END_RUNG wire#w2
   // the same network as SCL:
   #"AV-01.08"(LOCK := #lock,   // "Valve"
               LIOP_SEL := #Init,
               L_AUT := #Init,
               L_REMOTE := #Init,
               L_RESET := #Reset,
               FB_OPEN := #"AV-01.08".QCMD_OP,
               FB_CLOSE := NOT #"AV-01.08".QCMD_OP,
               L_MON := #Init,
               INSTANCE := 'AV-01.08');
END_REGION

REGION Network 9: AV-01.09
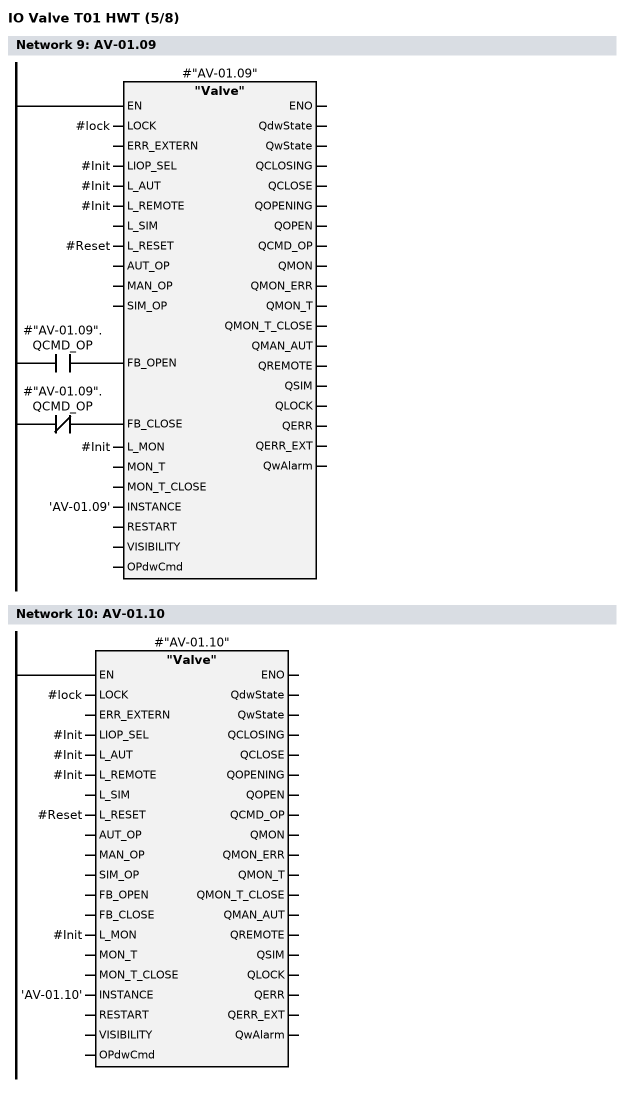
   RUNG wire#powerrail
      #"AV-01.09"(FB_OPEN := wire#w1, FB_CLOSE := wire#w2, LOCK := #lock, ERR_EXTERN :=, LIOP_SEL := #Init, L_AUT := #Init, L_REMOTE := #Init, L_SIM :=, L_RESET := #Reset, AUT_OP :=, MAN_OP :=, SIM_OP :=, L_MON := #Init, MON_T :=, MON_T_CLOSE :=, INSTANCE := 'AV-01.09', RESTART :=, VISIBILITY :=, OPdwCmd :=, QdwState =>, QwState =>, QCLOSING =>, QCLOSE =>, QOPENING =>, QOPEN =>, QCMD_OP =>, QMON =>, QMON_ERR =>, QMON_T =>, QMON_T_CLOSE =>, QMAN_AUT =>, QREMOTE =>, QSIM =>, QLOCK =>, QERR =>, QERR_EXT =>, QwAlarm =>)
   END_RUNG
   RUNG wire#powerrail
      Contact( #"AV-01.09".QCMD_OP )
   END_RUNG wire#w1
   RUNG wire#powerrail
      I_Contact( #"AV-01.09".QCMD_OP )
   END_RUNG wire#w2
   // the same network as SCL:
   #"AV-01.09"(LOCK := #lock,   // "Valve"
               LIOP_SEL := #Init,
               L_AUT := #Init,
               L_REMOTE := #Init,
               L_RESET := #Reset,
               FB_OPEN := #"AV-01.09".QCMD_OP,
               FB_CLOSE := NOT #"AV-01.09".QCMD_OP,
               L_MON := #Init,
               INSTANCE := 'AV-01.09');
END_REGION

REGION Network 10: AV-01.10
   RUNG wire#powerrail
      #"AV-01.10"(LOCK := #lock, ERR_EXTERN :=, LIOP_SEL := #Init, L_AUT := #Init, L_REMOTE := #Init, L_SIM :=, L_RESET := #Reset, AUT_OP :=, MAN_OP :=, SIM_OP :=, FB_OPEN :=, FB_CLOSE :=, L_MON := #Init, MON_T :=, MON_T_CLOSE :=, INSTANCE := 'AV-01.10', RESTART :=, VISIBILITY :=, OPdwCmd :=, QdwState =>, QwState =>, QCLOSING =>, QCLOSE =>, QOPENING =>, QOPEN =>, QCMD_OP =>, QMON =>, QMON_ERR =>, QMON_T =>, QMON_T_CLOSE =>, QMAN_AUT =>, QREMOTE =>, QSIM =>, QLOCK =>, QERR =>, QERR_EXT =>, QwAlarm =>)
   END_RUNG
   // the same network as SCL:
   #"AV-01.10"(LOCK := #lock,   // "Valve"
               LIOP_SEL := #Init,
               L_AUT := #Init,
               L_REMOTE := #Init,
               L_RESET := #Reset,
               L_MON := #Init,
               INSTANCE := 'AV-01.10');
END_REGION

REGION Network 11: AV-01.11
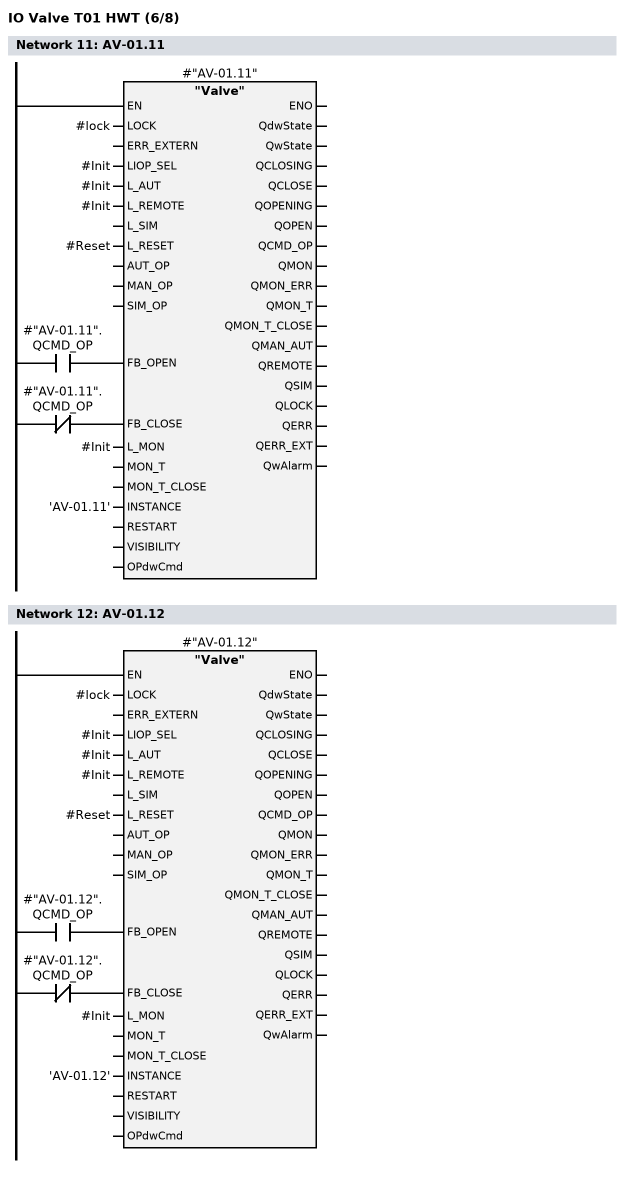
   RUNG wire#powerrail
      #"AV-01.11"(FB_OPEN := wire#w1, FB_CLOSE := wire#w2, LOCK := #lock, ERR_EXTERN :=, LIOP_SEL := #Init, L_AUT := #Init, L_REMOTE := #Init, L_SIM :=, L_RESET := #Reset, AUT_OP :=, MAN_OP :=, SIM_OP :=, L_MON := #Init, MON_T :=, MON_T_CLOSE :=, INSTANCE := 'AV-01.11', RESTART :=, VISIBILITY :=, OPdwCmd :=, QdwState =>, QwState =>, QCLOSING =>, QCLOSE =>, QOPENING =>, QOPEN =>, QCMD_OP =>, QMON =>, QMON_ERR =>, QMON_T =>, QMON_T_CLOSE =>, QMAN_AUT =>, QREMOTE =>, QSIM =>, QLOCK =>, QERR =>, QERR_EXT =>, QwAlarm =>)
   END_RUNG
   RUNG wire#powerrail
      Contact( #"AV-01.11".QCMD_OP )
   END_RUNG wire#w1
   RUNG wire#powerrail
      I_Contact( #"AV-01.11".QCMD_OP )
   END_RUNG wire#w2
   // the same network as SCL:
   #"AV-01.11"(LOCK := #lock,   // "Valve"
               LIOP_SEL := #Init,
               L_AUT := #Init,
               L_REMOTE := #Init,
               L_RESET := #Reset,
               FB_OPEN := #"AV-01.11".QCMD_OP,
               FB_CLOSE := NOT #"AV-01.11".QCMD_OP,
               L_MON := #Init,
               INSTANCE := 'AV-01.11');
END_REGION

REGION Network 12: AV-01.12
   RUNG wire#powerrail
      #"AV-01.12"(FB_OPEN := wire#w1, FB_CLOSE := wire#w2, LOCK := #lock, ERR_EXTERN :=, LIOP_SEL := #Init, L_AUT := #Init, L_REMOTE := #Init, L_SIM :=, L_RESET := #Reset, AUT_OP :=, MAN_OP :=, SIM_OP :=, L_MON := #Init, MON_T :=, MON_T_CLOSE :=, INSTANCE := 'AV-01.12', RESTART :=, VISIBILITY :=, OPdwCmd :=, QdwState =>, QwState =>, QCLOSING =>, QCLOSE =>, QOPENING =>, QOPEN =>, QCMD_OP =>, QMON =>, QMON_ERR =>, QMON_T =>, QMON_T_CLOSE =>, QMAN_AUT =>, QREMOTE =>, QSIM =>, QLOCK =>, QERR =>, QERR_EXT =>, QwAlarm =>)
   END_RUNG
   RUNG wire#powerrail
      Contact( #"AV-01.12".QCMD_OP )
   END_RUNG wire#w1
   RUNG wire#powerrail
      I_Contact( #"AV-01.12".QCMD_OP )
   END_RUNG wire#w2
   // the same network as SCL:
   #"AV-01.12"(LOCK := #lock,   // "Valve"
               LIOP_SEL := #Init,
               L_AUT := #Init,
               L_REMOTE := #Init,
               L_RESET := #Reset,
               FB_OPEN := #"AV-01.12".QCMD_OP,
               FB_CLOSE := NOT #"AV-01.12".QCMD_OP,
               L_MON := #Init,
               INSTANCE := 'AV-01.12');
END_REGION

REGION Network 13: AV-01.13
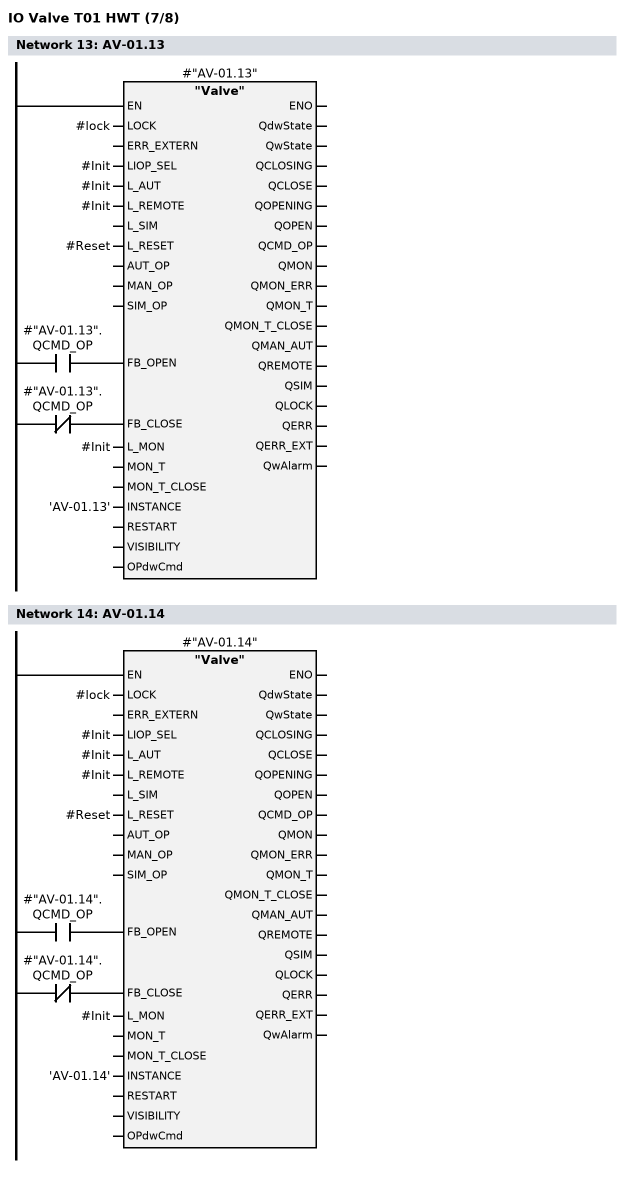
   RUNG wire#powerrail
      #"AV-01.13"(FB_OPEN := wire#w1, FB_CLOSE := wire#w2, LOCK := #lock, ERR_EXTERN :=, LIOP_SEL := #Init, L_AUT := #Init, L_REMOTE := #Init, L_SIM :=, L_RESET := #Reset, AUT_OP :=, MAN_OP :=, SIM_OP :=, L_MON := #Init, MON_T :=, MON_T_CLOSE :=, INSTANCE := 'AV-01.13', RESTART :=, VISIBILITY :=, OPdwCmd :=, QdwState =>, QwState =>, QCLOSING =>, QCLOSE =>, QOPENING =>, QOPEN =>, QCMD_OP =>, QMON =>, QMON_ERR =>, QMON_T =>, QMON_T_CLOSE =>, QMAN_AUT =>, QREMOTE =>, QSIM =>, QLOCK =>, QERR =>, QERR_EXT =>, QwAlarm =>)
   END_RUNG
   RUNG wire#powerrail
      Contact( #"AV-01.13".QCMD_OP )
   END_RUNG wire#w1
   RUNG wire#powerrail
      I_Contact( #"AV-01.13".QCMD_OP )
   END_RUNG wire#w2
   // the same network as SCL:
   #"AV-01.13"(LOCK := #lock,   // "Valve"
               LIOP_SEL := #Init,
               L_AUT := #Init,
               L_REMOTE := #Init,
               L_RESET := #Reset,
               FB_OPEN := #"AV-01.13".QCMD_OP,
               FB_CLOSE := NOT #"AV-01.13".QCMD_OP,
               L_MON := #Init,
               INSTANCE := 'AV-01.13');
END_REGION

REGION Network 14: AV-01.14
   RUNG wire#powerrail
      #"AV-01.14"(FB_OPEN := wire#w1, FB_CLOSE := wire#w2, LOCK := #lock, ERR_EXTERN :=, LIOP_SEL := #Init, L_AUT := #Init, L_REMOTE := #Init, L_SIM :=, L_RESET := #Reset, AUT_OP :=, MAN_OP :=, SIM_OP :=, L_MON := #Init, MON_T :=, MON_T_CLOSE :=, INSTANCE := 'AV-01.14', RESTART :=, VISIBILITY :=, OPdwCmd :=, QdwState =>, QwState =>, QCLOSING =>, QCLOSE =>, QOPENING =>, QOPEN =>, QCMD_OP =>, QMON =>, QMON_ERR =>, QMON_T =>, QMON_T_CLOSE =>, QMAN_AUT =>, QREMOTE =>, QSIM =>, QLOCK =>, QERR =>, QERR_EXT =>, QwAlarm =>)
   END_RUNG
   RUNG wire#powerrail
      Contact( #"AV-01.14".QCMD_OP )
   END_RUNG wire#w1
   RUNG wire#powerrail
      I_Contact( #"AV-01.14".QCMD_OP )
   END_RUNG wire#w2
   // the same network as SCL:
   #"AV-01.14"(LOCK := #lock,   // "Valve"
               LIOP_SEL := #Init,
               L_AUT := #Init,
               L_REMOTE := #Init,
               L_RESET := #Reset,
               FB_OPEN := #"AV-01.14".QCMD_OP,
               FB_CLOSE := NOT #"AV-01.14".QCMD_OP,
               L_MON := #Init,
               INSTANCE := 'AV-01.14');
END_REGION

REGION Network 15: AV-01.15
